C07328=1170.878,119.531,-53.606,-178.796,6.384,148.806
C07329=1170.873,119.780,-53.625,-178.793,6.386,148.805
C07330=1170.868,120.030,-53.645,-178.791,6.387,148.805
C07331=1170.864,120.279,-53.664,-178.789,6.388,148.804
C07332=1170.859,120.528,-53.683,-178.785,6.390,148.804
C07333=1170.854,120.778,-53.703,-178.783,6.391,148.803
C07334=1170.849,121.026,-53.722,-178.780,6.393,148.803
C07335=1170.844,121.276,-53.742,-178.777,6.395,148.803
C07336=1170.840,121.525,-53.761,-178.775,6.396,148.802
C07337=1170.835,121.774,-53.781,-178.772,6.397,148.802
C07338=1170.830,122.023,-53.800,-178.769,6.399,148.801
C07339=1170.826,122.273,-53.820,-178.766,6.401,148.801
C07340=1170.820,122.522,-53.839,-178.764,6.401,148.800
C07341=1170.816,122.771,-53.859,-178.761,6.403,148.800
C07342=1170.811,123.020,-53.878,-178.758,6.405,148.799
C07343=1170.806,123.269,-53.897,-178.756,6.406,148.799
C07344=1170.801,123.519,-53.917,-178.753,6.408,148.799
C07345=1170.796,123.767,-53.937,-178.751,6.409,148.798
C07346=1170.792,124.017,-53.957,-178.748,6.410,148.798
C07347=1170.787,124.266,-53.976,-178.745,6.412,148.797
C07348=1170.782,124.515,-53.995,-178.742,6.414,148.797
C07349=1170.778,124.764,-54.015,-178.740,6.415,148.796
C07350=1170.773,125.013,-54.035,-178.737,6.416,148.796
C07351=1170.768,125.263,-54.055,-178.734,6.418,148.795
C07352=1170.763,125.512,-54.074,-178.732,6.419,148.795
C07353=1170.758,125.761,-54.094,-178.729,6.421,148.795
C07354=1170.754,126.010,-54.114,-178.726,6.423,148.794
C07355=1170.749,126.259,-54.133,-178.723,6.425,148.794
C07356=1170.744,126.509,-54.153,-178.721,6.425,148.793
C07357=1170.739,126.758,-54.173,-178.718,6.427,148.793
C07358=1170.735,127.007,-54.193,-178.715,6.429,148.792
C07359=1170.729,127.256,-54.212,-178.713,6.430,148.792
C07360=1170.725,127.505,-54.233,-178.710,6.432,148.792
C07361=1170.720,127.755,-54.252,-178.708,6.433,148.791
C07362=1170.715,128.004,-54.272,-178.705,6.434,148.791
C07363=1170.710,128.252,-54.292,-178.702,6.436,148.790
C07364=1170.706,128.502,-54.312,-178.699,6.438,148.790
C07365=1170.701,128.752,-54.331,-178.697,6.440,148.789
C07366=1170.696,129.000,-54.352,-178.694,6.441,148.789
C07367=1170.691,129.249,-54.371,-178.692,6.442,148.789
C07368=1170.687,129.498,-54.391,-178.689,6.444,148.788
C07369=1170.682,129.748,-54.411,-178.686,6.445,148.788
C07370=1170.677,129.997,-54.431,-178.683,6.447,148.787
C07371=1170.672,130.246,-54.451,-178.680,6.449,148.787
C07372=1170.667,130.495,-54.470,-178.678,6.451,148.786
C07373=1170.663,130.744,-54.491,-178.675,6.452,148.786
C07374=1170.658,130.994,-54.510,-178.672,6.453,148.785
C07375=1170.654,131.243,-54.531,-178.670,6.455,148.785
C07376=1170.648,131.492,-54.550,-178.667,6.456,148.785
C07377=1170.643,131.741,-54.571,-178.664,6.458,148.784
C07378=1170.638,132.009,-54.592,-178.662,6.460,148.784
C07379=1170.633,132.278,-54.613,-178.658,6.461,148.783
C07380=1170.628,132.546,-54.635,-178.656,6.463,148.783
C07381=1170.623,132.815,-54.656,-178.653,6.465,148.782
C07382=1170.618,133.064,-54.677,-178.650,6.466,148.782
C07383=1170.613,133.314,-54.697,-178.647,6.468,148.781
C07384=1170.609,133.563,-54.717,-178.644,6.470,148.781
C07385=1170.604,133.812,-54.737,-178.642,6.471,148.781
C07386=1170.599,134.061,-54.757,-178.639,6.473,148.780
C07387=1170.595,134.310,-54.778,-178.637,6.474,148.780
C07388=1170.589,134.560,-54.798,-178.634,6.476,148.779
C07389=1170.585,134.809,-54.818,-178.631,6.477,148.779
C07390=1170.580,135.057,-54.839,-178.628,6.479,148.778
C07391=1170.575,135.307,-54.858,-178.626,6.481,148.778
C07392=1170.571,135.556,-54.879,-178.623,6.482,148.778
C07393=1170.566,135.805,-54.900,-178.620,6.484,148.777
C07394=1170.560,136.054,-54.919,-178.618,6.486,148.777
C07395=1170.556,136.303,-54.939,-178.615,6.488,148.776
C07396=1170.552,136.552,-54.960,-178.613,6.488,148.776
C07397=1170.546,136.802,-54.980,-178.610,6.490,148.775
C07398=1170.542,137.051,-55.000,-178.607,6.492,148.775
C07399=1170.537,137.300,-55.021,-178.604,6.493,148.775
C07400=1170.533,137.549,-55.041,-178.601,6.495,148.774
C07401=1170.528,137.798,-55.062,-178.599,6.497,148.774
C07402=1170.523,138.048,-55.082,-178.596,6.499,148.773
C07403=1170.518,138.296,-55.102,-178.593,6.500,148.773
C07404=1170.514,138.545,-55.122,-178.591,6.502,148.773
C07405=1170.509,138.795,-55.143,-178.588,6.503,148.772
C07406=1170.504,139.044,-55.164,-178.585,6.504,148.772
C07407=1170.500,139.293,-55.183,-178.583,6.506,148.771
C07408=1170.494,139.542,-55.204,-178.580,6.508,148.771
C07409=1170.489,139.791,-55.224,-178.577,6.510,148.771
C07410=1170.485,140.040,-55.245,-178.575,6.511,148.770
C07411=1170.480,140.289,-55.266,-178.572,6.513,148.770
C07412=1170.475,140.538,-55.286,-178.569,6.515,148.769
C07413=1170.471,140.787,-55.306,-178.566,6.517,148.769
C07414=1170.466,141.036,-55.327,-178.564,6.518,148.769
C07415=1170.461,141.286,-55.347,-178.561,6.520,148.768
C07416=1170.456,141.535,-55.368,-178.558,6.521,148.768
C07417=1170.451,141.784,-55.388,-178.556,6.522,148.767
C07418=1170.447,142.033,-55.409,-178.553,6.524,148.767
C07419=1170.442,142.282,-55.430,-178.550,6.526,148.766
C07420=1170.437,142.531,-55.450,-178.548,6.528,148.766
C07421=1170.432,142.780,-55.471,-178.545,6.529,148.766
C07422=1170.428,143.029,-55.491,-178.542,6.531,148.765
C07423=1170.424,143.279,-55.512,-178.540,6.533,148.765
C07424=1170.419,143.528,-55.533,-178.537,6.535,148.765
C07425=1170.414,143.777,-55.553,-178.534,6.536,148.764
C07426=1170.409,144.026,-55.574,-178.531,6.538,148.764
C07427=1170.405,144.275,-55.595,-178.528,6.539,148.763
C07428=1170.400,144.525,-55.616,-178.526,6.541,148.763
C07429=1170.395,144.773,-55.637,-178.523,6.543,148.762
C07430=1170.390,145.022,-55.658,-178.520,6.545,148.762
C07431=1170.386,145.271,-55.678,-178.517,6.546,148.762
C07432=1170.381,145.520,-55.699,-178.515,6.548,148.761
C07433=1170.376,145.769,-55.719,-178.513,6.549,148.761
C07434=1170.371,146.019,-55.740,-178.510,6.551,148.760
C07435=1170.367,146.268,-55.761,-178.507,6.553,148.760
C07436=1170.361,146.517,-55.782,-178.505,6.554,148.760
C07437=1170.357,146.765,-55.803,-178.502,6.556,148.759
C07438=1170.353,147.015,-55.824,-178.499,6.558,148.759
C07439=1170.348,147.264,-55.845,-178.496,6.560,148.759
C07440=1170.343,147.513,-55.866,-178.494,6.561,148.758
C07441=1170.338,147.763,-55.887,-178.491,6.563,148.758
C07442=1170.334,148.011,-55.908,-178.488,6.565,148.757
C07443=1170.329,148.260,-55.929,-178.485,6.566,148.757
C07444=1170.324,148.509,-55.949,-178.483,6.568,148.756
C07445=1170.319,148.758,-55.970,-178.480,6.570,148.756
C07446=1170.315,149.008,-55.992,-178.477,6.571,148.756
C07447=1170.310,149.257,-56.012,-178.474,6.573,148.755
C07448=1170.305,149.506,-56.033,-178.472,6.575,148.755
C07449=1170.301,149.755,-56.054,-178.469,6.577,148.754
C07450=1170.296,150.003,-56.075,-178.466,6.578,148.754
C07451=1170.291,150.253,-56.096,-178.464,6.580,148.754
C07452=1170.286,150.502,-56.117,-178.461,6.582,148.753
C07453=1170.282,150.751,-56.139,-178.458,6.584,148.753
C07454=1170.277,151.000,-56.160,-178.456,6.585,148.753
C07455=1170.272,151.249,-56.180,-178.453,6.587,148.752
C07456=1170.267,151.498,-56.202,-178.450,6.589,148.752
C07457=1170.262,151.747,-56.223,-178.447,6.591,148.751
C07458=1170.258,151.996,-56.245,-178.445,6.592,148.751
C07459=1170.254,152.245,-56.265,-178.442,6.594,148.751
C07460=1170.248,152.495,-56.286,-178.439,6.596,148.750
C07461=1170.244,152.743,-56.308,-178.437,6.598,148.750
C07462=1170.239,152.992,-56.328,-178.434,6.599,148.750
C07463=1170.235,153.242,-56.350,-178.431,6.601,148.749
C07464=1170.230,153.491,-56.371,-178.429,6.603,148.749
C07465=1170.225,153.740,-56.393,-178.426,6.605,148.748
C07466=1170.220,153.988,-56.413,-178.423,6.606,148.748
C07467=1170.216,154.238,-56.435,-178.421,6.608,148.748
C07468=1170.211,154.487,-56.456,-178.418,6.610,148.747
C07469=1170.206,154.736,-56.478,-178.415,6.612,148.747
C07470=1170.201,154.985,-56.499,-178.412,6.613,148.747
C07471=1170.197,155.234,-56.520,-178.410,6.615,148.746
C07472=1170.192,155.483,-56.541,-178.407,6.617,148.746
C07473=1170.187,155.732,-56.563,-178.404,6.619,148.745
C07474=1170.182,155.981,-56.584,-178.402,6.620,148.745
C07475=1170.178,156.230,-56.606,-178.399,6.622,148.745
C07476=1170.173,156.480,-56.627,-178.396,6.624,148.744
C07477=1170.169,156.728,-56.648,-178.394,6.626,148.744
C07478=1170.164,156.977,-56.670,-178.391,6.627,148.744
C07479=1170.159,157.227,-56.691,-178.388,6.629,148.743
C07480=1170.154,157.475,-56.713,-178.386,6.631,148.743
C07481=1170.149,157.724,-56.734,-178.383,6.633,148.742
C07482=1170.145,157.993,-56.757,-178.380,6.635,148.742
C07483=1170.139,158.262,-56.781,-178.377,6.637,148.742
C07484=1170.134,158.531,-56.803,-178.374,6.638,148.741
C07485=1170.129,158.800,-56.827,-178.371,6.640,148.741
C07486=1170.124,159.049,-56.848,-178.368,6.643,148.740
C07487=1170.120,159.299,-56.870,-178.365,6.644,148.740
C07488=1170.115,159.547,-56.892,-178.362,6.646,148.740
C07489=1170.111,159.796,-56.913,-178.360,6.648,148.739
C07490=1170.106,160.046,-56.935,-178.357,6.650,148.739
C07491=1170.101,160.294,-56.956,-178.355,6.652,148.739
C07492=1170.096,160.543,-56.978,-178.352,6.654,148.738
C07493=1170.092,160.792,-57.000,-178.349,6.655,148.738
C07494=1170.087,161.041,-57.022,-178.347,6.657,148.738
C07495=1170.083,161.291,-57.043,-178.344,6.659,148.737
C07496=1170.078,161.540,-57.065,-178.341,6.661,148.737
C07497=1170.073,161.788,-57.086,-178.339,6.662,148.736
C07498=1170.069,162.038,-57.108,-178.336,6.664,148.736
C07499=1170.064,162.286,-57.130,-178.333,6.666,148.736
C07500=1170.060,162.536,-57.152,-178.331,6.668,148.735
C07501=1170.054,162.785,-57.173,-178.328,6.669,148.735
C07502=1170.050,163.033,-57.195,-178.325,6.672,148.735
C07503=1170.045,163.283,-57.217,-178.322,6.674,148.734
C07504=1170.040,163.531,-57.238,-178.319,6.675,148.734
C07505=1170.036,163.781,-57.261,-178.317,6.677,148.733
C07506=1170.031,164.029,-57.282,-178.314,6.679,148.733
C07507=1170.026,164.279,-57.305,-178.311,6.681,148.733
C07508=1170.021,164.528,-57.327,-178.308,6.682,148.732
C07509=1170.016,164.776,-57.348,-178.306,6.684,148.732
C07510=1170.012,165.026,-57.370,-178.304,6.686,148.732
C07511=1170.007,165.274,-57.392,-178.301,6.688,148.731
C07512=1170.003,165.524,-57.414,-178.298,6.690,148.731
C07513=1169.998,165.772,-57.436,-178.296,6.692,148.731
C07514=1169.994,166.022,-57.458,-178.292,6.694,148.730
C07515=1169.989,166.270,-57.479,-178.290,6.696,148.730
C07516=1169.985,166.520,-57.501,-178.287,6.698,148.730
C07517=1169.979,166.769,-57.524,-178.284,6.699,148.729
C07518=1169.975,167.018,-57.546,-178.281,6.701,148.729
C07519=1169.970,167.267,-57.567,-178.279,6.703,148.729
C07520=1169.966,167.516,-57.590,-178.276,6.705,148.728
C07521=1169.961,167.765,-57.611,-178.273,6.706,148.728
C07522=1169.956,168.014,-57.634,-178.271,6.709,148.728
C07523=1169.951,168.262,-57.656,-178.268,6.711,148.727
C07524=1169.947,168.512,-57.678,-178.265,6.713,148.727
C07525=1169.942,168.760,-57.700,-178.263,6.715,148.727
C07526=1169.938,169.010,-57.722,-178.260,6.716,148.726
C07527=1169.932,169.258,-57.744,-178.257,6.718,148.726
C07528=1169.928,169.508,-57.766,-178.255,6.720,148.725
C07529=1169.924,169.756,-57.789,-178.252,6.722,148.725
C07530=1169.919,170.005,-57.811,-178.249,6.723,148.725
C07531=1169.914,170.254,-57.833,-178.246,6.726,148.724
C07532=1169.909,170.503,-57.855,-178.244,6.728,148.724
C07533=1169.905,170.752,-57.877,-178.241,6.730,148.724
C07534=1169.901,171.001,-57.900,-178.238,6.732,148.724
C07535=1169.896,171.250,-57.922,-178.236,6.733,148.723
C07536=1169.891,171.499,-57.944,-178.233,6.735,148.723
C07537=1169.887,171.748,-57.967,-178.230,6.737,148.722
C07538=1169.881,171.997,-57.989,-178.228,6.739,148.722
C07539=1169.877,172.246,-58.011,-178.224,6.741,148.722
C07540=1169.872,172.495,-58.033,-178.222,6.743,148.721
C07541=1169.867,172.744,-58.056,-178.219,6.745,148.721
C07542=1169.863,172.993,-58.078,-178.217,6.747,148.721
C07543=1169.858,173.242,-58.100,-178.214,6.749,148.720
C07544=1169.853,173.491,-58.123,-178.211,6.750,148.720
C07545=1169.849,173.740,-58.145,-178.209,6.752,148.720
C07546=1169.845,173.988,-58.168,-178.205,6.755,148.719
C07547=1169.840,174.238,-58.190,-178.203,6.757,148.719
C07548=1169.835,174.486,-58.212,-178.201,6.759,148.719
C07549=1169.830,174.735,-58.235,-178.198,6.760,148.719
C07550=1169.826,174.985,-58.257,-178.195,6.762,148.718
C07551=1169.821,175.233,-58.280,-178.192,6.764,148.718
C07552=1169.816,175.483,-58.302,-178.189,6.767,148.717
C07553=1169.812,175.731,-58.325,-178.187,6.768,148.717
C07554=1169.807,175.980,-58.347,-178.184,6.770,148.717
C07555=1169.803,176.229,-58.370,-178.182,6.772,148.717
C07556=1169.798,176.479,-58.393,-178.179,6.774,148.716
C07557=1169.793,176.727,-58.415,-178.176,6.776,148.716
C07558=1169.789,176.976,-58.437,-178.173,6.778,148.715
C07559=1169.784,177.225,-58.461,-178.170,6.780,148.715
C07560=1169.779,177.474,-58.482,-178.168,6.782,148.715
C07561=1169.775,177.723,-58.506,-178.165,6.784,148.715
C07562=1169.770,177.972,-58.528,-178.163,6.786,148.714
C07563=1169.765,178.220,-58.551,-178.160,6.788,148.714
C07564=1169.761,178.469,-58.573,-178.157,6.790,148.714
C07565=1169.756,178.719,-58.596,-178.154,6.792,148.713
C07566=1169.752,178.967,-58.619,-178.151,6.794,148.713
C07567=1169.746,179.216,-58.641,-178.149,6.796,148.713
C07568=1169.742,179.465,-58.664,-178.147,6.797,148.712
C07569=1169.738,179.714,-58.687,-178.143,6.800,148.712
C07570=1169.733,179.964,-58.710,-178.141,6.802,148.712
C07571=1169.728,180.212,-58.732,-178.138,6.804,148.711
C07572=1169.724,180.461,-58.756,-178.135,6.805,148.711
C07573=1169.719,180.710,-58.778,-178.133,6.807,148.711
C07574=1169.715,180.959,-58.801,-178.130,6.810,148.710
C07575=1169.710,181.207,-58.823,-178.127,6.812,148.710
C07576=1169.705,181.456,-58.847,-178.124,6.814,148.710
C07577=1169.700,181.706,-58.869,-178.122,6.815,148.709
C07578=1169.696,181.955,-58.892,-178.119,6.818,148.709
C07579=1169.691,182.203,-58.915,-178.116,6.820,148.709
C07580=1169.687,182.452,-58.938,-178.114,6.822,148.709
C07581=1169.682,182.701,-58.961,-178.111,6.824,148.708
C07582=1169.677,182.950,-58.984,-178.108,6.825,148.708
C07583=1169.673,183.199,-59.007,-178.105,6.828,148.708
C07584=1169.669,183.448,-59.030,-178.103,6.830,148.707
C07585=1169.663,183.696,-59.053,-178.100,6.832,148.707
C07586=1169.659,183.966,-59.078,-178.097,6.834,148.707
C07587=1169.653,184.236,-59.103,-178.094,6.836,148.706
C07588=1169.648,184.505,-59.128,-178.091,6.839,148.706
C07589=1169.644,184.775,-59.152,-178.088,6.840,148.706
C07590=1169.639,185.024,-59.175,-178.086,6.843,148.705
C07591=1169.634,185.273,-59.199,-178.083,6.845,148.705
C07592=1169.629,185.522,-59.222,-178.080,6.847,148.705
C07593=1169.626,185.771,-59.245,-178.077,6.849,148.704
C07594=1169.621,186.020,-59.268,-178.075,6.850,148.704
C07595=1169.616,186.269,-59.292,-178.073,6.853,148.704
C07596=1169.611,186.517,-59.315,-178.069,6.855,148.704
C07597=1169.607,186.766,-59.337,-178.067,6.857,148.703
C07598=1169.602,187.015,-59.361,-178.064,6.859,148.703
C07599=1169.597,187.264,-59.384,-178.062,6.861,148.703
C07600=1169.593,187.513,-59.407,-178.058,6.863,148.702
C07601=1169.589,187.762,-59.430,-178.056,6.865,148.702
C07602=1169.584,188.011,-59.454,-178.053,6.867,148.702
C07603=1169.579,188.260,-59.477,-178.051,6.869,148.702
C07604=1169.575,188.509,-59.500,-178.048,6.872,148.701
C07605=1169.569,188.757,-59.523,-178.045,6.873,148.701
C07606=1169.565,189.006,-59.547,-178.042,6.875,148.701
C07607=1169.561,189.255,-59.569,-178.040,6.878,148.700
C07608=1169.556,189.504,-59.593,-178.037,6.880,148.700
C07609=1169.552,189.752,-59.617,-178.034,6.882,148.700
C07610=1169.547,190.001,-59.640,-178.032,6.883,148.699
C07611=1169.542,190.250,-59.664,-178.029,6.886,148.699
C07612=1169.538,190.499,-59.687,-178.026,6.888,148.699
C07613=1169.533,190.748,-59.710,-178.023,6.890,148.699
C07614=1169.528,190.997,-59.734,-178.021,6.892,148.698
C07615=1169.523,191.246,-59.757,-178.018,6.895,148.698
C07616=1169.520,191.495,-59.780,-178.015,6.896,148.698
C07617=1169.515,191.744,-59.804,-178.013,6.898,148.697
C07618=1169.510,191.993,-59.827,-178.010,6.901,148.697
C07619=1169.506,192.242,-59.851,-178.007,6.903,148.697
C07620=1169.501,192.490,-59.875,-178.004,6.905,148.697
C07621=1169.497,192.739,-59.898,-178.002,6.906,148.696
C07622=1169.492,192.988,-59.921,-177.999,6.909,148.696
C07623=1169.487,193.237,-59.945,-177.996,6.911,148.696
C07624=1169.483,193.486,-59.969,-177.994,6.913,148.695
C07625=1169.478,193.735,-59.992,-177.991,6.916,148.695
C07626=1169.473,193.984,-60.015,-177.988,6.918,148.695
C07627=1169.469,194.232,-60.040,-177.986,6.919,148.695
C07628=1169.464,194.481,-60.063,-177.983,6.921,148.694
C07629=1169.460,194.730,-60.086,-177.980,6.924,148.694
C07630=1169.455,194.978,-60.110,-177.977,6.926,148.694
C07631=1169.451,195.228,-60.134,-177.975,6.928,148.693
C07632=1169.446,195.476,-60.158,-177.972,6.931,148.693
C07633=1169.441,195.725,-60.181,-177.969,6.932,148.693
C07634=1169.437,195.974,-60.204,-177.967,6.934,148.693
C07635=1169.432,196.222,-60.229,-177.964,6.937,148.692
C07636=1169.427,196.472,-60.253,-177.961,6.939,148.692
C07637=1169.422,196.720,-60.277,-177.958,6.941,148.692
C07638=1169.418,196.969,-60.300,-177.955,6.943,148.691
C07639=1169.413,197.218,-60.324,-177.953,6.945,148.691
C07640=1169.409,197.467,-60.347,-177.950,6.947,148.691
C07641=1169.405,197.716,-60.372,-177.947,6.950,148.691
C07642=1169.400,197.965,-60.395,-177.945,6.952,148.691
C07643=1169.396,198.213,-60.419,-177.942,6.954,148.690
C07644=1169.391,198.462,-60.443,-177.939,6.956,148.690
C07645=1169.386,198.711,-60.467,-177.937,6.958,148.690
C07646=1169.381,198.960,-60.491,-177.934,6.960,148.689
C07647=1169.377,199.208,-60.515,-177.931,6.963,148.689
C07648=1169.372,199.457,-60.538,-177.929,6.965,148.689
C07649=1169.368,199.706,-60.562,-177.926,6.967,148.689
C07650=1169.364,199.955,-60.587,-177.923,6.969,148.688
C07651=1169.359,200.204,-60.611,-177.921,6.971,148.688
C07652=1169.354,200.453,-60.635,-177.918,6.973,148.688
C07653=1169.350,200.701,-60.659,-177.915,6.976,148.687
C07654=1169.345,200.950,-60.682,-177.912,6.978,148.687
C07655=1169.341,201.199,-60.706,-177.910,6.980,148.687
C07656=1169.336,201.448,-60.731,-177.907,6.982,148.687
C07657=1169.331,201.697,-60.755,-177.904,6.984,148.687
C07658=1169.327,201.945,-60.779,-177.902,6.986,148.686
C07659=1169.323,202.194,-60.803,-177.899,6.989,148.686
C07660=1169.317,202.443,-60.827,-177.896,6.991,148.686
C07661=1169.313,202.692,-60.851,-177.894,6.993,148.685
C07662=1169.309,202.941,-60.875,-177.891,6.996,148.685
C07663=1169.305,203.189,-60.899,-177.888,6.997,148.685
C07664=1169.299,203.438,-60.923,-177.885,7.000,148.685
C07665=1169.295,203.687,-60.947,-177.883,7.002,148.685
C07666=1169.290,203.935,-60.971,-177.880,7.004,148.684
C07667=1169.286,204.185,-60.996,-177.877,7.007,148.684
C07668=1169.281,204.433,-61.020,-177.875,7.009,148.684
C07669=1169.277,204.682,-61.045,-177.872,7.010,148.683
C07670=1169.272,204.931,-61.068,-177.869,7.013,148.683
C07671=1169.268,205.180,-61.093,-177.866,7.015,148.683
C07672=1169.263,205.428,-61.117,-177.863,7.018,148.683
C07673=1169.258,205.677,-61.142,-177.861,7.020,148.682
C07674=1169.254,205.926,-61.166,-177.858,7.022,148.682
C07675=1169.249,206.175,-61.191,-177.856,7.024,148.682
C07676=1169.245,206.423,-61.215,-177.853,7.026,148.682
C07677=1169.241,206.672,-61.239,-177.850,7.028,148.681
C07678=1169.236,206.921,-61.264,-177.847,7.031,148.681
C07679=1169.232,207.170,-61.288,-177.845,7.033,148.681
C07680=1169.226,207.419,-61.312,-177.842,7.036,148.681
C07681=1169.222,207.667,-61.336,-177.839,7.037,148.680
C07682=1169.217,207.917,-61.361,-177.837,7.039,148.680
C07683=1169.213,208.165,-61.385,-177.834,7.042,148.680
C07684=1169.209,208.414,-61.409,-177.831,7.044,148.680
C07685=1169.204,208.662,-61.435,-177.828,7.047,148.680
C07686=1169.200,208.911,-61.459,-177.826,7.049,148.679
C07687=1169.195,209.160,-61.484,-177.823,7.050,148.679
C07688=1169.190,209.408,-61.508,-177.820,7.053,148.679
C07689=1169.186,209.657,-61.533,-177.818,7.055,148.678
C07690=1169.181,209.928,-61.560,-177.815,7.058,148.678
C07691=1169.175,210.198,-61.586,-177.812,7.061,148.678
C07692=1169.171,210.469,-61.613,-177.809,7.063,148.678
C07693=1169.166,210.739,-61.639,-177.806,7.065,148.677
C07694=1169.162,210.989,-61.664,-177.803,7.068,148.677
C07695=1169.157,211.237,-61.689,-177.800,7.070,148.677
C07696=1169.153,211.485,-61.713,-177.798,7.072,148.677
C07697=1169.148,211.735,-61.738,-177.795,7.075,148.677
C07698=1169.143,211.983,-61.763,-177.793,7.077,148.676
C07699=1169.138,212.232,-61.787,-177.789,7.079,148.676
C07700=1169.134,212.480,-61.813,-177.787,7.081,148.676
C07701=1169.130,212.729,-61.837,-177.784,7.084,148.676
C07702=1169.125,212.978,-61.862,-177.781,7.086,148.675
C07703=1169.121,213.227,-61.886,-177.779,7.088,148.675
C07704=1169.116,213.475,-61.911,-177.776,7.091,148.675
C07705=1169.112,213.724,-61.936,-177.774,7.093,148.675
C07706=1169.107,213.973,-61.960,-177.770,7.095,148.674
C07707=1169.103,214.222,-61.985,-177.768,7.097,148.674
C07708=1169.098,214.470,-62.011,-177.765,7.100,148.674
C07709=1169.093,214.719,-62.035,-177.763,7.102,148.674
C07710=1169.089,214.968,-62.060,-177.760,7.105,148.674
C07711=1169.084,215.216,-62.085,-177.757,7.107,148.674
C07712=1169.080,215.465,-62.110,-177.755,7.109,148.673
C07713=1169.075,215.714,-62.134,-177.752,7.111,148.673
C07714=1169.071,215.963,-62.160,-177.749,7.113,148.673
C07715=1169.067,216.211,-62.184,-177.746,7.116,148.672
C07716=1169.062,216.460,-62.210,-177.744,7.118,148.672
C07717=1169.057,216.709,-62.235,-177.741,7.121,148.672
C07718=1169.053,216.958,-62.260,-177.738,7.123,148.672
C07719=1169.049,217.206,-62.285,-177.735,7.125,148.672
C07720=1169.044,217.455,-62.310,-177.733,7.128,148.671
C07721=1169.039,217.703,-62.335,-177.730,7.130,148.671
C07722=1169.035,217.953,-62.360,-177.728,7.132,148.671
C07723=1169.031,218.201,-62.385,-177.724,7.135,148.671
C07724=1169.026,218.450,-62.410,-177.722,7.137,148.671
C07725=1169.021,218.698,-62.435,-177.719,7.140,148.670
C07726=1169.017,218.948,-62.460,-177.717,7.142,148.670
C07727=1169.012,219.196,-62.486,-177.714,7.144,148.670
C07728=1169.008,219.445,-62.510,-177.711,7.147,148.670
C07729=1169.003,219.693,-62.535,-177.709,7.148,148.669
C07730=1168.999,219.942,-62.561,-177.706,7.151,148.669
C07731=1168.994,220.190,-62.586,-177.703,7.153,148.669
C07732=1168.990,220.439,-62.612,-177.700,7.156,148.669
C07733=1168.985,220.688,-62.636,-177.698,7.158,148.669
C07734=1168.981,220.936,-62.661,-177.695,7.161,148.669
C07735=1168.977,221.185,-62.687,-177.692,7.163,148.668
C07736=1168.972,221.434,-62.712,-177.690,7.165,148.668
C07737=1168.967,221.683,-62.738,-177.687,7.167,148.668
C07738=1168.963,221.931,-62.763,-177.684,7.170,148.668
C07739=1168.958,222.180,-62.788,-177.681,7.172,148.667
C07740=1168.953,222.428,-62.813,-177.679,7.175,148.667
C07741=1168.949,222.677,-62.839,-177.677,7.177,148.667
C07742=1168.945,222.926,-62.865,-177.673,7.180,148.667
C07743=1168.940,223.175,-62.890,-177.671,7.182,148.667
C07744=1168.936,223.423,-62.915,-177.668,7.184,148.666
C07745=1168.931,223.671,-62.940,-177.666,7.187,148.666
C07746=1168.927,223.920,-62.966,-177.662,7.189,148.666
C07747=1168.923,224.170,-62.991,-177.660,7.192,148.666
C07748=1168.918,224.418,-63.016,-177.657,7.194,148.666
C07749=1168.914,224.666,-63.042,-177.654,7.197,148.665
C07750=1168.909,224.915,-63.068,-177.652,7.199,148.665
C07751=1168.905,225.163,-63.093,-177.649,7.202,148.665
C07752=1168.900,225.412,-63.119,-177.647,7.204,148.665
C07753=1168.896,225.662,-63.144,-177.643,7.206,148.665
C07754=1168.891,225.910,-63.169,-177.641,7.208,148.665
C07755=1168.887,226.159,-63.195,-177.638,7.211,148.664
C07756=1168.883,226.407,-63.221,-177.636,7.213,148.664
C07757=1168.877,226.656,-63.247,-177.633,7.216,148.664
C07758=1168.873,226.905,-63.273,-177.630,7.218,148.664
C07759=1168.869,227.153,-63.298,-177.628,7.221,148.664
C07760=1168.864,227.401,-63.324,-177.625,7.223,148.663
C07761=1168.859,227.650,-63.349,-177.622,7.226,148.663
C07762=1168.855,227.899,-63.375,-177.619,7.228,148.663
C07763=1168.850,228.147,-63.401,-177.617,7.230,148.663
C07764=1168.846,228.396,-63.426,-177.614,7.233,148.663
C07765=1168.842,228.645,-63.452,-177.611,7.235,148.662
C07766=1168.838,228.894,-63.478,-177.609,7.238,148.662
C07767=1168.832,229.142,-63.504,-177.606,7.240,148.662
C07768=1168.828,229.391,-63.530,-177.603,7.243,148.662
C07769=1168.824,229.640,-63.555,-177.600,7.245,148.662
C07770=1168.819,229.888,-63.581,-177.598,7.248,148.662
C07771=1168.815,230.137,-63.606,-177.595,7.251,148.661
C07772=1168.810,230.385,-63.632,-177.592,7.252,148.661
C07773=1168.806,230.634,-63.658,-177.590,7.255,148.661
C07774=1168.801,230.883,-63.684,-177.587,7.257,148.661
C07775=1168.797,231.131,-63.710,-177.584,7.260,148.661
C07776=1168.793,231.380,-63.736,-177.582,7.262,148.661
C07777=1168.788,231.628,-63.762,-177.579,7.265,148.660
C07778=1168.783,231.877,-63.788,-177.576,7.268,148.660
C07779=1168.778,232.126,-63.814,-177.574,7.270,148.660
C07780=1168.774,232.374,-63.839,-177.571,7.272,148.660
C07781=1168.770,232.623,-63.866,-177.568,7.275,148.660
C07782=1168.765,232.872,-63.892,-177.565,7.277,148.659
C07783=1168.761,233.120,-63.918,-177.563,7.279,148.659
C07784=1168.756,233.369,-63.943,-177.560,7.282,148.659
C07785=1168.752,233.617,-63.970,-177.557,7.285,148.659
C07786=1168.747,233.866,-63.996,-177.555,7.287,148.659
C07787=1168.743,234.115,-64.022,-177.552,7.290,148.659
C07788=1168.739,234.364,-64.048,-177.549,7.292,148.658
C07789=1168.734,234.612,-64.075,-177.547,7.295,148.658
C07790=1168.730,234.860,-64.100,-177.544,7.298,148.658
C07791=1168.725,235.109,-64.126,-177.541,7.299,148.658
C07792=1168.721,235.357,-64.153,-177.538,7.302,148.658
C07793=1168.716,235.606,-64.179,-177.536,7.305,148.658
C07794=1168.712,235.877,-64.207,-177.533,7.307,148.657
C07795=1168.707,236.150,-64.236,-177.530,7.310,148.657
C07796=1168.702,236.421,-64.265,-177.527,7.313,148.657
C07797=1168.698,236.693,-64.293,-177.524,7.316,148.657
C07798=1168.693,236.941,-64.320,-177.521,7.318,148.657
C07799=1168.688,237.189,-64.345,-177.519,7.320,148.657
C07800=1168.683,237.438,-64.372,-177.516,7.323,148.656
C07801=1168.679,237.687,-64.398,-177.513,7.326,148.656
C07802=1168.675,237.935,-64.425,-177.511,7.328,148.656
C07803=1168.670,238.184,-64.451,-177.508,7.331,148.656
C07804=1168.666,238.432,-64.477,-177.505,7.334,148.656
C07805=1168.661,238.681,-64.504,-177.502,7.336,148.656
C07806=1168.657,238.930,-64.530,-177.500,7.339,148.656
C07807=1168.653,239.179,-64.557,-177.498,7.341,148.655
C07808=1168.649,239.427,-64.583,-177.494,7.344,148.655
C07809=1168.644,239.676,-64.609,-177.492,7.347,148.655
C07810=1168.640,239.924,-64.636,-177.489,7.349,148.655
C07811=1168.635,240.173,-64.662,-177.487,7.352,148.655
C07812=1168.630,240.421,-64.688,-177.483,7.354,148.655
C07813=1168.626,240.669,-64.715,-177.481,7.356,148.655
C07814=1168.621,240.918,-64.741,-177.478,7.359,148.654
C07815=1168.617,241.167,-64.768,-177.475,7.362,148.654
C07816=1168.613,241.415,-64.795,-177.473,7.364,148.654
C07817=1168.608,241.664,-64.821,-177.470,7.367,148.654
C07818=1168.603,241.912,-64.848,-177.467,7.370,148.654
C07819=1168.599,242.161,-64.875,-177.465,7.372,148.654
C07820=1168.594,242.410,-64.901,-177.462,7.375,148.654
C07821=1168.590,242.658,-64.927,-177.459,7.378,148.653
C07822=1168.586,242.906,-64.954,-177.457,7.380,148.653
C07823=1168.582,243.155,-64.981,-177.454,7.382,148.653
C07824=1168.577,243.404,-65.007,-177.452,7.385,148.653
C07825=1168.572,243.652,-65.034,-177.449,7.388,148.653
C07826=1168.568,243.900,-65.061,-177.446,7.390,148.653
C07827=1168.564,244.149,-65.088,-177.444,7.392,148.653
C07828=1168.559,244.397,-65.115,-177.441,7.395,148.652
C07829=1168.555,244.647,-65.141,-177.438,7.398,148.652
C07830=1168.551,244.895,-65.168,-177.435,7.401,148.652
C07831=1168.546,245.144,-65.195,-177.433,7.403,148.652
C07832=1168.542,245.392,-65.222,-177.430,7.406,148.652
C07833=1168.537,245.640,-65.249,-177.427,7.409,148.652
C07834=1168.533,245.889,-65.276,-177.425,7.411,148.652
C07835=1168.529,246.137,-65.302,-177.422,7.414,148.651
C07836=1168.524,246.386,-65.328,-177.419,7.417,148.651
C07837=1168.519,246.635,-65.356,-177.417,7.419,148.651
C07838=1168.515,246.883,-65.382,-177.414,7.422,148.651
C07839=1168.511,247.131,-65.409,-177.411,7.425,148.651
C07840=1168.506,247.380,-65.436,-177.409,7.426,148.651
C07841=1168.501,247.628,-65.463,-177.406,7.429,148.651
C07842=1168.498,247.877,-65.490,-177.403,7.432,148.651
C07843=1168.493,248.126,-65.517,-177.401,7.434,148.651
C07844=1168.489,248.374,-65.544,-177.398,7.437,148.651
C07845=1168.484,248.623,-65.571,-177.395,7.440,148.650
C07846=1168.479,248.871,-65.598,-177.392,7.443,148.650
C07847=1168.475,249.120,-65.625,-177.390,7.445,148.650
C07848=1168.471,249.368,-65.652,-177.387,7.448,148.650
C07849=1168.466,249.616,-65.679,-177.384,7.451,148.650
C07850=1168.462,249.865,-65.707,-177.382,7.453,148.650
C07851=1168.458,250.114,-65.734,-177.379,7.456,148.650
C07852=1168.454,250.362,-65.761,-177.376,7.459,148.650
C07853=1168.449,250.610,-65.788,-177.374,7.461,148.649
C07854=1168.445,250.859,-65.815,-177.371,7.464,148.649
C07855=1168.440,251.107,-65.842,-177.369,7.467,148.649
C07856=1168.436,251.356,-65.869,-177.365,7.469,148.649
C07857=1168.431,251.604,-65.897,-177.363,7.472,148.649
C07858=1168.427,251.853,-65.924,-177.360,7.475,148.649
C07859=1168.422,252.101,-65.951,-177.358,7.478,148.649
C07860=1168.418,252.349,-65.978,-177.355,7.480,148.649
C07861=1168.414,252.599,-66.005,-177.353,7.483,148.649
C07862=1168.410,252.847,-66.033,-177.350,7.485,148.648
C07863=1168.405,253.095,-66.060,-177.347,7.488,148.648
C07864=1168.401,253.344,-66.087,-177.345,7.490,148.648
C07865=1168.396,253.593,-66.114,-177.342,7.493,148.648
C07866=1168.392,253.841,-66.142,-177.339,7.496,148.648
C07867=1168.387,254.089,-66.169,-177.336,7.499,148.648
C07868=1168.383,254.338,-66.196,-177.334,7.501,148.648
C07869=1168.379,254.586,-66.224,-177.331,7.504,148.648
C07870=1168.374,254.835,-66.251,-177.328,7.507,148.648
C07871=1168.370,255.083,-66.278,-177.325,7.510,148.648
C07872=1168.365,255.331,-66.306,-177.323,7.512,148.647
C07873=1168.361,255.580,-66.334,-177.320,7.515,148.647
C07874=1168.357,255.828,-66.361,-177.318,7.518,148.647
C07875=1168.352,256.077,-66.388,-177.315,7.521,148.647
C07876=1168.348,256.325,-66.416,-177.313,7.523,148.647
C07877=1168.344,256.574,-66.444,-177.310,7.526,148.647
C07878=1168.339,256.822,-66.471,-177.307,7.529,148.647
C07879=1168.335,257.070,-66.499,-177.304,7.532,148.647
C07880=1168.331,257.319,-66.526,-177.302,7.534,148.647
C07881=1168.326,257.567,-66.554,-177.299,7.537,148.647
C07882=1168.321,257.816,-66.581,-177.296,7.540,148.647
C07883=1168.317,258.065,-66.610,-177.294,7.543,148.646
C07884=1168.313,258.313,-66.637,-177.291,7.545,148.646
C07885=1168.308,258.561,-66.664,-177.289,7.548,148.646
C07886=1168.304,258.810,-66.692,-177.286,7.551,148.646
C07887=1168.300,259.058,-66.720,-177.283,7.554,148.646
C07888=1168.296,259.306,-66.747,-177.281,7.555,148.646
C07889=1168.291,259.555,-66.775,-177.278,7.558,148.646
C07890=1168.286,259.803,-66.803,-177.275,7.561,148.646
C07891=1168.282,260.052,-66.830,-177.272,7.564,148.646
C07892=1168.278,260.300,-66.858,-177.269,7.567,148.646
C07893=1168.274,260.548,-66.886,-177.267,7.569,148.646
C07894=1168.269,260.797,-66.913,-177.265,7.572,148.646
C07895=1168.265,261.046,-66.942,-177.262,7.575,148.645
C07896=1168.260,261.293,-66.970,-177.259,7.578,148.645
C07897=1168.256,261.543,-66.997,-177.257,7.580,148.645
C07898=1168.251,261.815,-67.027,-177.254,7.584,148.645
C07899=1168.246,262.089,-67.058,-177.251,7.587,148.645
C07900=1168.242,262.361,-67.090,-177.248,7.590,148.645
C07901=1168.237,262.635,-67.120,-177.245,7.593,148.645
C07902=1168.233,262.883,-67.147,-177.242,7.596,148.645
C07903=1168.228,263.132,-67.176,-177.239,7.599,148.645
C07904=1168.224,263.380,-67.204,-177.237,7.602,148.645
C07905=1168.219,263.628,-67.232,-177.234,7.604,148.645
C07906=1168.216,263.876,-67.260,-177.232,7.607,148.645
C07907=1168.210,264.125,-67.287,-177.229,7.610,148.645
C07908=1168.206,264.374,-67.315,-177.226,7.613,148.645
C07909=1168.202,264.622,-67.343,-177.223,7.616,148.644
C07910=1168.198,264.870,-67.372,-177.221,7.618,148.644
C07911=1168.193,265.118,-67.400,-177.218,7.621,148.644
C07912=1168.189,265.367,-67.429,-177.216,7.624,148.644
C07913=1168.184,265.615,-67.456,-177.213,7.627,148.644
C07914=1168.181,265.864,-67.484,-177.210,7.630,148.644
C07915=1168.176,266.112,-67.513,-177.208,7.632,148.644
C07916=1168.171,266.360,-67.541,-177.205,7.635,148.644
C07917=1168.167,266.609,-67.568,-177.203,7.638,148.644
C07918=1168.162,266.857,-67.596,-177.200,7.641,148.644
C07919=1168.158,267.106,-67.625,-177.197,7.644,148.644
C07920=1168.154,267.355,-67.653,-177.195,7.646,148.644
C07921=1168.149,267.602,-67.681,-177.192,7.649,148.644
C07922=1168.145,267.851,-67.710,-177.189,7.652,148.644
C07923=1168.141,268.099,-67.738,-177.187,7.655,148.644
C07924=1168.137,268.347,-67.766,-177.184,7.658,148.644
C07925=1168.132,268.595,-67.795,-177.181,7.661,148.644
C07926=1168.128,268.844,-67.823,-177.179,7.663,148.643
C07927=1168.123,269.092,-67.851,-177.176,7.666,148.643
C07928=1168.120,269.341,-67.879,-177.173,7.669,148.643
C07929=1168.114,269.589,-67.908,-177.171,7.672,148.643
C07930=1168.111,269.837,-67.936,-177.168,7.675,148.643
C07931=1168.106,270.086,-67.964,-177.165,7.678,148.643
C07932=1168.102,270.334,-67.992,-177.163,7.680,148.643
C07933=1168.098,270.583,-68.022,-177.160,7.683,148.643
C07934=1168.093,270.830,-68.050,-177.157,7.686,148.643
C07935=1168.089,271.079,-68.078,-177.155,7.689,148.643
C07936=1168.084,271.327,-68.107,-177.152,7.692,148.643
C07937=1168.080,271.576,-68.135,-177.150,7.695,148.643
C07938=1168.076,271.824,-68.164,-177.147,7.698,148.643
C07939=1168.071,272.072,-68.192,-177.145,7.700,148.643
C07940=1168.067,272.321,-68.221,-177.142,7.703,148.643
C07941=1168.063,272.569,-68.249,-177.139,7.706,148.643
C07942=1168.058,272.817,-68.278,-177.136,7.709,148.643
C07943=1168.054,273.066,-68.307,-177.134,7.712,148.643
C07944=1168.050,273.314,-68.335,-177.131,7.715,148.643
C07945=1168.045,273.562,-68.364,-177.128,7.718,148.643
C07946=1168.041,273.811,-68.393,-177.126,7.720,148.643
C07947=1168.037,274.059,-68.421,-177.123,7.723,148.643
C07948=1168.032,274.307,-68.450,-177.121,7.726,148.642
C07949=1168.028,274.556,-68.479,-177.118,7.729,148.642
C07950=1168.024,274.803,-68.507,-177.116,7.732,148.643
C07951=1168.019,275.052,-68.536,-177.113,7.735,148.643
C07952=1168.015,275.301,-68.565,-177.110,7.738,148.643
C07953=1168.011,275.548,-68.593,-177.108,7.740,148.642
C07954=1168.006,275.797,-68.622,-177.105,7.743,148.642
C07955=1168.002,276.046,-68.651,-177.102,7.746,148.642
C07956=1167.998,276.294,-68.680,-177.100,7.749,148.642
C07957=1167.994,276.542,-68.709,-177.097,7.752,148.642
C07958=1167.989,276.791,-68.737,-177.094,7.755,148.642
C07959=1167.985,277.039,-68.767,-177.092,7.758,148.642
C07960=1167.981,277.287,-68.795,-177.089,7.761,148.642
C07961=1167.976,277.535,-68.824,-177.087,7.763,148.642
C07962=1167.972,277.784,-68.853,-177.084,7.766,148.642
C07963=1167.968,278.032,-68.882,-177.081,7.769,148.642
C07964=1167.963,278.280,-68.910,-177.079,7.772,148.642
C07965=1167.959,278.528,-68.940,-177.076,7.775,148.642
C07966=1167.955,278.777,-68.969,-177.073,7.778,148.642
C07967=1167.951,279.026,-68.998,-177.071,7.782,148.642
C07968=1167.946,279.273,-69.027,-177.068,7.784,148.642
C07969=1167.942,279.521,-69.056,-177.065,7.787,148.642
C07970=1167.938,279.770,-69.084,-177.063,7.790,148.642
C07971=1167.934,280.018,-69.114,-177.060,7.793,148.642
C07972=1167.930,280.266,-69.143,-177.058,7.796,148.642
C07973=1167.924,280.515,-69.172,-177.055,7.798,148.642
C07974=1167.920,280.763,-69.201,-177.053,7.802,148.642
C07975=1167.916,281.011,-69.231,-177.050,7.805,148.642
C07976=1167.912,281.260,-69.259,-177.047,7.808,148.642
C07977=1167.908,281.508,-69.288,-177.044,7.811,148.642
C07978=1167.903,281.756,-69.317,-177.042,7.814,148.642
C07979=1167.899,282.004,-69.347,-177.039,7.817,148.642
C07980=1167.895,282.252,-69.376,-177.037,7.820,148.642
C07981=1167.890,282.501,-69.405,-177.034,7.822,148.642
C07982=1167.886,282.749,-69.434,-177.032,7.825,148.642
C07983=1167.882,282.997,-69.463,-177.029,7.828,148.642
C07984=1167.877,283.245,-69.493,-177.026,7.831,148.642
C07985=1167.873,283.493,-69.522,-177.023,7.834,148.642
C07986=1167.869,283.742,-69.552,-177.021,7.837,148.642
C07987=1167.864,283.991,-69.581,-177.018,7.840,148.642
C07988=1167.860,284.239,-69.610,-177.016,7.843,148.642
C07989=1167.856,284.487,-69.639,-177.013,7.846,148.642
C07990=1167.851,284.735,-69.669,-177.010,7.849,148.642
C07991=1167.847,284.983,-69.698,-177.008,7.852,148.642
C07992=1167.843,285.231,-69.727,-177.005,7.855,148.642
C07993=1167.839,285.479,-69.757,-177.003,7.857,148.642
C07994=1167.835,285.728,-69.786,-177.000,7.860,148.642
C07995=1167.830,285.976,-69.816,-176.997,7.863,148.642
C07996=1167.826,286.224,-69.845,-176.995,7.867,148.642
C07997=1167.822,286.472,-69.875,-176.992,7.870,148.642
C07998=1167.818,286.721,-69.904,-176.990,7.873,148.642
C07999=1167.813,286.969,-69.934,-176.987,7.876,148.642
C08000=1167.809,287.218,-69.964,-176.984,7.879,148.642
C08001=1167.804,287.465,-69.993,-176.982,7.882,148.642
C08002=1167.799,287.740,-70.026,-176.979,7.885,148.642
C08003=1167.795,288.015,-70.058,-176.976,7.889,148.642
C08004=1167.791,288.290,-70.091,-176.973,7.892,148.642
C08005=1167.786,288.565,-70.124,-176.970,7.895,148.642
C08006=1167.781,288.813,-70.153,-176.968,7.898,148.642
C08007=1167.777,289.062,-70.183,-176.965,7.901,148.642
C08008=1167.773,289.309,-70.213,-176.963,7.904,148.642
C08009=1167.768,289.558,-70.243,-176.960,7.907,148.642
C08010=1167.764,289.806,-70.273,-176.958,7.910,148.642
C08011=1167.760,290.054,-70.302,-176.955,7.913,148.642
C08012=1167.756,290.303,-70.332,-176.952,7.916,148.642
C08013=1167.752,290.550,-70.362,-176.949,7.919,148.642
C08014=1167.747,290.799,-70.392,-176.947,7.922,148.642
C08015=1167.743,291.047,-70.421,-176.944,7.925,148.642
C08016=1167.739,291.295,-70.451,-176.942,7.928,148.642
C08017=1167.735,291.543,-70.481,-176.939,7.931,148.642
C08018=1167.730,291.792,-70.511,-176.937,7.934,148.642
C08019=1167.726,292.040,-70.540,-176.934,7.937,148.642
C08020=1167.722,292.288,-70.570,-176.931,7.940,148.642
C08021=1167.718,292.536,-70.600,-176.928,7.943,148.642
C08022=1167.713,292.784,-70.630,-176.926,7.947,148.642
C08023=1167.709,293.032,-70.660,-176.923,7.950,148.642
C08024=1167.705,293.280,-70.690,-176.920,7.953,148.642
C08025=1167.700,293.529,-70.720,-176.918,7.956,148.643
C08026=1167.696,293.777,-70.750,-176.915,7.959,148.642
C08027=1167.692,294.025,-70.779,-176.913,7.962,148.642
C08028=1167.687,294.273,-70.810,-176.910,7.965,148.643
C08029=1167.684,294.522,-70.840,-176.908,7.968,148.643
C08030=1167.680,294.769,-70.870,-176.906,7.970,148.643
C08031=1167.675,295.018,-70.900,-176.903,7.973,148.642
C08032=1167.671,295.266,-70.930,-176.900,7.977,148.643
C08033=1167.667,295.514,-70.960,-176.898,7.980,148.643
C08034=1167.662,295.762,-70.990,-176.895,7.982,148.643
C08035=1167.658,296.010,-71.020,-176.893,7.986,148.643
C08036=1167.653,296.258,-71.051,-176.890,7.989,148.643
C08037=1167.649,296.506,-71.080,-176.887,7.992,148.643
C08038=1167.646,296.755,-71.111,-176.885,7.995,148.643
C08039=1167.641,297.003,-71.141,-176.882,7.998,148.643
C08040=1167.637,297.251,-71.171,-176.879,8.001,148.643
C08041=1167.632,297.499,-71.202,-176.877,8.004,148.643
C08042=1167.628,297.747,-71.231,-176.874,8.007,148.643
C08043=1167.624,297.995,-71.262,-176.872,8.010,148.643
C08044=1167.620,298.243,-71.292,-176.869,8.013,148.643
C08045=1167.615,298.492,-71.322,-176.867,8.016,148.643
C08046=1167.612,298.740,-71.353,-176.864,8.019,148.643
C08047=1167.607,298.988,-71.383,-176.862,8.023,148.643
C08048=1167.603,299.236,-71.413,-176.859,8.026,148.643
C08049=1167.598,299.484,-71.444,-176.856,8.029,148.643
C08050=1167.595,299.732,-71.474,-176.854,8.032,148.643
C08051=1167.590,299.981,-71.504,-176.851,8.035,148.643
C08052=1167.586,300.228,-71.534,-176.848,8.038,148.643
C08053=1167.581,300.476,-71.565,-176.846,8.041,148.644
C08054=1167.578,300.724,-71.595,-176.843,8.044,148.644
C08055=1167.574,300.973,-71.626,-176.841,8.047,148.644
C08056=1167.569,301.221,-71.656,-176.838,8.050,148.644
C08057=1167.565,301.469,-71.687,-176.836,8.053,148.644
C08058=1167.560,301.717,-71.717,-176.833,8.057,148.644
C08059=1167.556,301.965,-71.748,-176.831,8.060,148.644
C08060=1167.552,302.213,-71.779,-176.828,8.063,148.644
C08061=1167.548,302.461,-71.809,-176.825,8.066,148.644
C08062=1167.543,302.709,-71.839,-176.822,8.070,148.644
C08063=1167.539,302.957,-71.870,-176.820,8.073,148.644
C08064=1167.535,303.206,-71.901,-176.817,8.076,148.644
C08065=1167.531,303.454,-71.931,-176.814,8.079,148.644
C08066=1167.526,303.702,-71.962,-176.812,8.082,148.644
C08067=1167.522,303.950,-71.992,-176.809,8.085,148.644
C08068=1167.518,304.198,-72.023,-176.807,8.089,148.644
C08069=1167.514,304.446,-72.054,-176.804,8.092,148.644
C08070=1167.509,304.694,-72.085,-176.802,8.094,148.644
C08071=1167.506,304.942,-72.115,-176.799,8.098,148.645
C08072=1167.501,305.190,-72.146,-176.797,8.101,148.645
C08073=1167.497,305.438,-72.177,-176.794,8.104,148.645
C08074=1167.493,305.687,-72.208,-176.792,8.107,148.645
C08075=1167.489,305.934,-72.238,-176.789,8.110,148.645
C08076=1167.484,306.182,-72.269,-176.786,8.113,148.645
C08077=1167.480,306.431,-72.300,-176.784,8.116,148.645
C08078=1167.476,306.679,-72.331,-176.781,8.120,148.645
C08079=1167.471,306.926,-72.362,-176.779,8.123,148.645
C08080=1167.468,307.175,-72.393,-176.776,8.126,148.645
C08081=1167.463,307.423,-72.423,-176.774,8.129,148.645
C08082=1167.459,307.671,-72.454,-176.771,8.132,148.645
C08083=1167.455,307.919,-72.485,-176.769,8.135,148.645
C08084=1167.450,308.167,-72.516,-176.766,8.138,148.646
C08085=1167.447,308.414,-72.547,-176.764,8.141,148.646
C08086=1167.443,308.663,-72.578,-176.761,8.144,148.646
C08087=1167.438,308.911,-72.609,-176.759,8.148,148.646
C08088=1167.433,309.159,-72.640,-176.755,8.151,148.646
C08089=1167.430,309.407,-72.671,-176.753,8.155,148.646
C08090=1167.425,309.655,-72.702,-176.750,8.158,148.646
C08091=1167.421,309.904,-72.733,-176.748,8.161,148.646
C08092=1167.416,310.151,-72.764,-176.745,8.164,148.646
C08093=1167.413,310.398,-72.795,-176.743,8.167,148.646
C08094=1167.409,310.647,-72.826,-176.740,8.170,148.646
C08095=1167.404,310.895,-72.857,-176.738,8.173,148.646
C08096=1167.401,311.143,-72.889,-176.735,8.176,148.646
C08097=1167.396,311.391,-72.919,-176.733,8.180,148.647
C08098=1167.392,311.640,-72.951,-176.730,8.183,148.647
C08099=1167.388,311.887,-72.982,-176.728,8.186,148.647
C08100=1167.384,312.136,-73.013,-176.725,8.189,148.647
C08101=1167.379,312.383,-73.045,-176.723,8.192,148.647
C08102=1167.375,312.631,-73.075,-176.720,8.195,148.647
C08103=1167.371,312.879,-73.107,-176.718,8.199,148.647
C08104=1167.366,313.127,-73.138,-176.714,8.202,148.647
C08105=1167.362,313.376,-73.169,-176.712,8.206,148.647
C08106=1167.357,313.653,-73.204,-176.709,8.209,148.647
C08107=1167.353,313.929,-73.239,-176.707,8.213,148.648
C08108=1167.349,314.207,-73.275,-176.704,8.216,148.648
C08109=1167.344,314.484,-73.309,-176.701,8.220,148.648
C08110=1167.339,314.731,-73.341,-176.698,8.223,148.648
C08111=1167.336,314.979,-73.373,-176.696,8.226,148.648
C08112=1167.331,315.227,-73.403,-176.693,8.229,148.648
C08113=1167.327,315.475,-73.435,-176.691,8.232,148.648
C08114=1167.323,315.723,-73.466,-176.688,8.235,148.648
C08115=1167.319,315.971,-73.498,-176.686,8.239,148.648
C08116=1167.315,316.219,-73.529,-176.683,8.242,148.648
C08117=1167.310,316.468,-73.561,-176.680,8.246,148.649
C08118=1167.306,316.716,-73.593,-176.678,8.249,148.649
C08119=1167.302,316.963,-73.624,-176.675,8.252,148.649
C08120=1167.298,317.212,-73.655,-176.673,8.255,148.649
C08121=1167.294,317.459,-73.687,-176.670,8.258,148.649
C08122=1167.290,317.707,-73.719,-176.668,8.262,148.649
C08123=1167.285,317.955,-73.749,-176.665,8.265,148.649
C08124=1167.282,318.203,-73.781,-176.663,8.268,148.649
C08125=1167.277,318.451,-73.814,-176.661,8.271,148.649
C08126=1167.273,318.699,-73.845,-176.658,8.274,148.649
C08127=1167.269,318.947,-73.876,-176.655,8.278,148.650
C08128=1167.265,319.195,-73.908,-176.652,8.281,148.650
C08129=1167.261,319.443,-73.940,-176.650,8.285,148.650
C08130=1167.256,319.691,-73.972,-176.647,8.287,148.650
C08131=1167.252,319.939,-74.004,-176.645,8.291,148.650
C08132=1167.248,320.187,-74.035,-176.643,8.294,148.650
C08133=1167.244,320.435,-74.066,-176.640,8.297,148.650
C08134=1167.239,320.683,-74.099,-176.638,8.300,148.650
C08135=1167.236,320.931,-74.131,-176.634,8.304,148.650
C08136=1167.231,321.178,-74.162,-176.632,8.307,148.651
C08137=1167.228,321.426,-74.194,-176.630,8.311,148.651
C08138=1167.223,321.675,-74.226,-176.627,8.314,148.651
C08139=1167.219,321.922,-74.258,-176.625,8.317,148.651
C08140=1167.215,322.170,-74.290,-176.622,8.320,148.651
C08141=1167.211,322.418,-74.322,-176.620,8.323,148.651
C08142=1167.206,322.666,-74.354,-176.617,8.327,148.651
C08143=1167.203,322.914,-74.385,-176.614,8.330,148.651
C08144=1167.198,323.162,-74.418,-176.612,8.334,148.652
C08145=1167.195,323.410,-74.450,-176.610,8.337,148.652
C08146=1167.190,323.657,-74.481,-176.607,8.340,148.652
C08147=1167.186,323.906,-74.514,-176.605,8.343,148.652
C08148=1167.182,324.154,-74.545,-176.602,8.347,148.652
C08149=1167.178,324.401,-74.577,-176.599,8.350,148.652
C08150=1167.173,324.650,-74.609,-176.597,8.353,148.652
C08151=1167.170,324.898,-74.641,-176.594,8.357,148.653
C08152=1167.166,325.146,-74.673,-176.592,8.360,148.653
C08153=1167.161,325.393,-74.706,-176.589,8.363,148.653
C08154=1167.157,325.641,-74.738,-176.587,8.366,148.653
C08155=1167.153,325.889,-74.770,-176.584,8.369,148.653
C08156=1167.149,326.137,-74.802,-176.582,8.373,148.653
C08157=1167.144,326.385,-74.834,-176.580,8.376,148.653
C08158=1167.141,326.633,-74.866,-176.576,8.380,148.654
C08159=1167.136,326.880,-74.899,-176.574,8.383,148.654
C08160=1167.133,327.129,-74.931,-176.572,8.386,148.654
C08161=1167.128,327.376,-74.963,-176.570,8.390,148.654
C08162=1167.124,327.624,-74.995,-176.567,8.393,148.654
C08163=1167.120,327.872,-75.028,-176.565,8.396,148.654
C08164=1167.116,328.120,-75.060,-176.562,8.400,148.655
C08165=1167.111,328.368,-75.092,-176.559,8.403,148.655
C08166=1167.107,328.616,-75.124,-176.557,8.406,148.655
C08167=1167.103,328.863,-75.157,-176.554,8.410,148.655
C08168=1167.100,329.111,-75.189,-176.552,8.413,148.655
C08169=1167.095,329.360,-75.221,-176.549,8.416,148.655
C08170=1167.092,329.607,-75.254,-176.546,8.420,148.655
C08171=1167.087,329.855,-75.286,-176.544,8.423,148.656
C08172=1167.083,330.103,-75.319,-176.542,8.427,148.656
C08173=1167.079,330.351,-75.351,-176.539,8.430,148.656
C08174=1167.074,330.599,-75.383,-176.537,8.433,148.656
C08175=1167.071,330.846,-75.416,-176.535,8.436,148.656
C08176=1167.067,331.095,-75.448,-176.532,8.440,148.656
C08177=1167.062,331.342,-75.481,-176.529,8.443,148.656
C08178=1167.058,331.590,-75.513,-176.527,8.447,148.657
C08179=1167.054,331.838,-75.546,-176.524,8.450,148.657
C08180=1167.050,332.086,-75.578,-176.522,8.453,148.657
C08181=1167.046,332.333,-75.611,-176.519,8.456,148.657
C08182=1167.042,332.582,-75.643,-176.516,8.460,148.657
C08183=1167.038,332.829,-75.677,-176.514,8.464,148.658
C08184=1167.034,333.077,-75.708,-176.512,8.467,148.658
C08185=1167.029,333.324,-75.741,-176.510,8.470,148.658
C08186=1167.025,333.572,-75.774,-176.507,8.473,148.658
C08187=1167.021,333.820,-75.806,-176.504,8.477,148.658
C08188=1167.017,334.068,-75.839,-176.502,8.481,148.658
C08189=1167.013,334.316,-75.872,-176.499,8.484,148.659
C08190=1167.009,334.564,-75.905,-176.497,8.487,148.659
C08191=1167.005,334.811,-75.938,-176.494,8.490,148.659
C08192=1167.001,335.060,-75.970,-176.492,8.494,148.659
C08193=1166.997,335.308,-76.003,-176.489,8.498,148.659
C08194=1166.992,335.555,-76.036,-176.487,8.501,148.659
C08195=1166.989,335.803,-76.068,-176.485,8.504,148.660
C08196=1166.985,336.051,-76.101,-176.482,8.507,148.660
C08197=1166.980,336.299,-76.134,-176.479,8.511,148.660
C08198=1166.976,336.546,-76.168,-176.477,8.515,148.660
C08199=1166.972,336.795,-76.200,-176.474,8.518,148.660
C08200=1166.968,337.042,-76.233,-176.472,8.521,148.661
C08201=1166.964,337.290,-76.266,-176.470,8.524,148.661
C08202=1166.960,337.538,-76.299,-176.467,8.529,148.661
C08203=1166.956,337.785,-76.332,-176.465,8.532,148.661
C08204=1166.952,338.033,-76.365,-176.462,8.535,148.661
C08205=1166.947,338.282,-76.398,-176.460,8.538,148.661
C08206=1166.943,338.529,-76.431,-176.457,8.542,148.662
C08207=1166.940,338.777,-76.463,-176.455,8.546,148.662
C08208=1166.936,339.024,-76.497,-176.452,8.549,148.662
C08209=1166.932,339.272,-76.530,-176.450,8.552,148.662
C08210=1166.926,339.551,-76.567,-176.447,8.556,148.663
C08211=1166.922,339.831,-76.604,-176.444,8.560,148.663
C08212=1166.917,340.110,-76.642,-176.441,8.564,148.663
C08213=1166.912,340.390,-76.679,-176.439,8.568,148.663
C08214=1166.908,340.638,-76.712,-176.436,8.572,148.663
C08215=1166.904,340.886,-76.745,-176.434,8.575,148.664
C08216=1166.900,341.134,-76.778,-176.431,8.578,148.664
C08217=1166.896,341.381,-76.811,-176.429,8.581,148.664
C08218=1166.892,341.629,-76.845,-176.427,8.585,148.664
C08219=1166.888,341.876,-76.878,-176.424,8.589,148.664
C08220=1166.884,342.124,-76.912,-176.421,8.592,148.665
C08221=1166.880,342.372,-76.945,-176.419,8.595,148.665
C08222=1166.876,342.620,-76.978,-176.417,8.599,148.665
C08223=1166.872,342.868,-77.011,-176.414,8.603,148.665
C08224=1166.868,343.115,-77.045,-176.412,8.606,148.665
C08225=1166.864,343.363,-77.078,-176.409,8.609,148.666
C08226=1166.859,343.611,-77.111,-176.407,8.613,148.666
C08227=1166.855,343.859,-77.144,-176.404,8.617,148.666
C08228=1166.851,344.106,-77.178,-176.402,8.620,148.666
C08229=1166.847,344.353,-77.211,-176.400,8.623,148.667
C08230=1166.843,344.601,-77.244,-176.397,8.628,148.667
C08231=1166.840,344.850,-77.278,-176.395,8.631,148.667
C08232=1166.835,345.098,-77.311,-176.392,8.634,148.667
C08233=1166.831,345.345,-77.345,-176.390,8.637,148.667
C08234=1166.827,345.593,-77.379,-176.387,8.642,148.668
C08235=1166.823,345.840,-77.412,-176.385,8.645,148.668
C08236=1166.819,346.088,-77.445,-176.383,8.648,148.668
C08237=1166.815,346.336,-77.479,-176.380,8.651,148.668
C08238=1166.811,346.584,-77.512,-176.377,8.656,148.669
C08239=1166.806,346.832,-77.546,-176.375,8.659,148.669
C08240=1166.802,347.079,-77.580,-176.373,8.662,148.669
C08241=1166.798,347.326,-77.613,-176.370,8.666,148.669
C08242=1166.794,347.574,-77.646,-176.368,8.670,148.670
C08243=1166.791,347.822,-77.680,-176.365,8.673,148.670
C08244=1166.786,348.070,-77.714,-176.363,8.676,148.670
C08245=1166.782,348.317,-77.748,-176.361,8.681,148.670
C08246=1166.778,348.565,-77.781,-176.358,8.684,148.671
C08247=1166.774,348.813,-77.814,-176.356,8.687,148.671
C08248=1166.770,349.061,-77.849,-176.353,8.691,148.671
C08249=1166.766,349.308,-77.882,-176.351,8.695,148.671
C08250=1166.762,349.555,-77.916,-176.349,8.698,148.672
C08251=1166.758,349.803,-77.949,-176.346,8.701,148.672
C08252=1166.754,350.051,-77.984,-176.343,8.705,148.672
C08253=1166.750,350.299,-78.017,-176.341,8.709,148.672
C08254=1166.746,350.546,-78.051,-176.339,8.712,148.673
C08255=1166.741,350.794,-78.085,-176.336,8.716,148.673
C08256=1166.738,351.042,-78.119,-176.334,8.720,148.673
C08257=1166.734,351.289,-78.153,-176.332,8.723,148.673
C08258=1166.730,351.537,-78.186,-176.329,8.727,148.674
C08259=1166.726,351.785,-78.221,-176.327,8.730,148.674
C08260=1166.722,352.033,-78.254,-176.324,8.734,148.674
C08261=1166.717,352.280,-78.289,-176.322,8.738,148.675
C08262=1166.713,352.527,-78.323,-176.320,8.741,148.675
C08263=1166.710,352.776,-78.356,-176.317,8.745,148.675
C08264=1166.705,353.023,-78.391,-176.315,8.749,148.675
C08265=1166.701,353.270,-78.424,-176.312,8.752,148.675
C08266=1166.698,353.519,-78.458,-176.310,8.756,148.676
C08267=1166.693,353.766,-78.492,-176.308,8.760,148.676
C08268=1166.689,354.013,-78.526,-176.305,8.763,148.676
C08269=1166.686,354.261,-78.561,-176.303,8.766,148.677
C08270=1166.681,354.509,-78.594,-176.300,8.770,148.677
C08271=1166.677,354.756,-78.629,-176.298,8.774,148.677
C08272=1166.674,355.004,-78.663,-176.296,8.777,148.677
C08273=1166.669,355.252,-78.697,-176.293,8.781,148.678
C08274=1166.665,355.499,-78.731,-176.291,8.785,148.678
C08275=1166.662,355.747,-78.765,-176.289,8.788,148.678
C08276=1166.657,355.995,-78.799,-176.286,8.793,148.679
C08277=1166.654,356.242,-78.834,-176.284,8.796,148.679
C08278=1166.649,356.490,-78.868,-176.282,8.799,148.679
C08279=1166.645,356.737,-78.902,-176.279,8.804,148.680
C08280=1166.641,356.985,-78.937,-176.277,8.807,148.680
C08281=1166.638,357.232,-78.971,-176.274,8.810,148.680
C08282=1166.634,357.480,-79.005,-176.272,8.815,148.680
C08283=1166.629,357.728,-79.040,-176.270,8.818,148.681
C08284=1166.625,357.975,-79.074,-176.267,8.821,148.681
C08285=1166.621,358.224,-79.108,-176.265,8.826,148.681
C08286=1166.617,358.471,-79.142,-176.263,8.829,148.682
C08287=1166.613,358.719,-79.177,-176.260,8.833,148.682
C08288=1166.609,358.966,-79.210,-176.258,8.837,148.682
C08289=1166.606,359.213,-79.246,-176.256,8.840,148.682
C08290=1166.601,359.461,-79.280,-176.253,8.844,148.683
C08291=1166.598,359.709,-79.315,-176.251,8.848,148.683
C08292=1166.593,359.956,-79.349,-176.249,8.851,148.683
C08293=1166.590,360.204,-79.383,-176.246,8.855,148.684
C08294=1166.586,360.451,-79.418,-176.244,8.859,148.684
C08295=1166.581,360.699,-79.452,-176.241,8.863,148.684
C08296=1166.578,360.947,-79.487,-176.239,8.866,148.685
C08297=1166.573,361.194,-79.521,-176.237,8.870,148.685
C08298=1166.569,361.442,-79.556,-176.235,8.874,148.685
C08299=1166.566,361.689,-79.590,-176.232,8.877,148.686
C08300=1166.562,361.937,-79.625,-176.230,8.882,148.686
C08301=1166.558,362.185,-79.660,-176.228,8.885,148.686
C08302=1166.554,362.432,-79.694,-176.226,8.889,148.687
C08303=1166.550,362.680,-79.729,-176.223,8.893,148.687
C08304=1166.546,362.927,-79.764,-176.221,8.896,148.688
C08305=1166.542,363.175,-79.799,-176.219,8.900,148.688
C08306=1166.538,363.422,-79.833,-176.216,8.904,148.688
C08307=1166.534,363.670,-79.868,-176.214,8.908,148.689
C08308=1166.530,363.917,-79.903,-176.212,8.912,148.689
C08309=1166.526,364.165,-79.938,-176.210,8.915,148.689
C08310=1166.522,364.412,-79.971,-176.207,8.919,148.690
C08311=1166.518,364.660,-80.007,-176.205,8.923,148.690
C08312=1166.514,364.908,-80.042,-176.203,8.927,148.690
C08313=1166.510,365.155,-80.076,-176.201,8.930,148.691
C08314=1166.505,365.438,-80.116,-176.198,8.934,148.691
C08315=1166.501,365.720,-80.156,-176.196,8.939,148.692
C08316=1166.497,366.002,-80.196,-176.193,8.943,148.692
C08317=1166.492,366.284,-80.235,-176.191,8.948,148.693
C08318=1166.488,366.532,-80.270,-176.189,8.951,148.693
C08319=1166.484,366.780,-80.306,-176.187,8.956,148.693
C08320=1166.480,367.027,-80.340,-176.185,8.959,148.694
C08321=1166.476,367.274,-80.376,-176.183,8.963,148.694
C08322=1166.472,367.522,-80.409,-176.180,8.967,148.695
C08323=1166.469,367.769,-80.445,-176.178,8.971,148.695
C08324=1166.465,368.017,-80.480,-176.176,8.974,148.695
C08325=1166.460,368.264,-80.515,-176.175,8.978,148.696
C08326=1166.456,368.512,-80.550,-176.172,8.982,148.696
C08327=1166.453,368.760,-80.585,-176.170,8.986,148.697
C08328=1166.448,369.006,-80.621,-176.168,8.989,148.697
C08329=1166.444,369.255,-80.655,-176.167,8.993,148.698
C08330=1166.441,369.502,-80.691,-176.165,8.998,148.698
C08331=1166.436,369.749,-80.725,-176.163,9.001,148.699
C08332=1166.433,369.997,-80.761,-176.161,9.005,148.699
C08333=1166.429,370.244,-80.796,-176.159,9.009,148.700
C08334=1166.424,370.492,-80.831,-176.157,9.012,148.700
C08335=1166.421,370.739,-80.866,-176.155,9.016,148.700
C08336=1166.417,370.987,-80.902,-176.153,9.021,148.701
C08337=1166.412,371.234,-80.937,-176.151,9.024,148.702
C08338=1166.409,371.482,-80.972,-176.150,9.028,148.702
C08339=1166.405,371.729,-81.008,-176.148,9.032,148.703
C08340=1166.401,371.977,-81.042,-176.146,9.035,148.703
C08341=1166.397,372.224,-81.078,-176.144,9.039,148.703
C08342=1166.393,372.472,-81.113,-176.143,9.043,148.704
C08343=1166.389,372.719,-81.148,-176.141,9.046,148.705
C08344=1166.385,372.967,-81.183,-176.140,9.050,148.705
C08345=1166.381,373.214,-81.219,-176.138,9.054,148.706
C08346=1166.378,373.462,-81.254,-176.136,9.058,148.706
C08347=1166.373,373.708,-81.289,-176.135,9.061,148.707
C08348=1166.370,373.956,-81.325,-176.133,9.065,148.707
C08349=1166.366,374.204,-81.360,-176.132,9.069,148.708
C08350=1166.362,374.452,-81.395,-176.130,9.073,148.708
C08351=1166.358,374.698,-81.431,-176.128,9.077,148.709
C08352=1166.353,374.946,-81.467,-176.127,9.081,148.710
C08353=1166.350,375.194,-81.502,-176.125,9.084,148.710
C08354=1166.346,375.441,-81.538,-176.124,9.088,148.711
C08355=1166.342,375.688,-81.573,-176.122,9.092,148.711
C08356=1166.338,375.935,-81.609,-176.121,9.096,148.712
C08357=1166.334,376.184,-81.643,-176.120,9.099,148.712
C08358=1166.331,376.431,-81.679,-176.118,9.103,148.713
C08359=1166.326,376.679,-81.715,-176.117,9.107,148.713
C08360=1166.322,376.926,-81.750,-176.115,9.110,148.714
C08361=1166.318,377.173,-81.786,-176.114,9.114,148.715
C08362=1166.315,377.421,-81.821,-176.113,9.117,148.715
C08363=1166.311,377.668,-81.857,-176.112,9.121,148.716
C08364=1166.306,377.916,-81.893,-176.110,9.125,148.717
C08365=1166.302,378.163,-81.928,-176.109,9.129,148.717
C08366=1166.299,378.410,-81.964,-176.108,9.133,148.718
C08367=1166.295,378.658,-81.999,-176.107,9.136,148.719
C08368=1166.291,378.905,-82.035,-176.106,9.140,148.719
C08369=1166.287,379.153,-82.071,-176.105,9.143,148.720
C08370=1166.283,379.400,-82.106,-176.103,9.147,148.720
C08371=1166.279,379.647,-82.142,-176.103,9.151,148.721
C08372=1166.276,379.894,-82.178,-176.101,9.155,148.722
C08373=1166.271,380.142,-82.214,-176.101,9.158,148.722
C08374=1166.267,380.390,-82.250,-176.100,9.162,148.723
C08375=1166.264,380.637,-82.285,-176.099,9.165,148.724
C08376=1166.260,380.884,-82.320,-176.097,9.169,148.724
C08377=1166.255,381.132,-82.357,-176.097,9.172,148.725
C08378=1166.251,381.379,-82.392,-176.095,9.176,148.726
C08379=1166.248,381.627,-82.428,-176.095,9.180,148.727
C08380=1166.244,381.874,-82.465,-176.094,9.183,148.727
C08381=1166.240,382.121,-82.500,-176.093,9.187,148.728
C08382=1166.236,382.369,-82.536,-176.092,9.190,148.729
C08383=1166.232,382.616,-82.571,-176.092,9.193,148.729
C08384=1166.228,382.864,-82.607,-176.091,9.196,148.730
C08385=1166.224,383.111,-82.642,-176.090,9.201,148.731
C08386=1166.221,383.358,-82.679,-176.090,9.204,148.732
C08387=1166.216,383.606,-82.715,-176.089,9.207,148.732
C08388=1166.213,383.853,-82.750,-176.088,9.211,148.733
C08389=1166.209,384.101,-82.786,-176.088,9.214,148.734
C08390=1166.205,384.348,-82.823,-176.087,9.217,148.734
C08391=1166.201,384.595,-82.858,-176.086,9.221,148.735
C08392=1166.197,384.842,-82.894,-176.086,9.225,148.736
C08393=1166.193,385.090,-82.930,-176.085,9.228,148.737
C08394=1166.189,385.337,-82.966,-176.085,9.231,148.737
C08395=1166.185,385.585,-83.002,-176.085,9.234,148.738
C08396=1166.181,385.832,-83.038,-176.084,9.237,148.739
C08397=1166.178,386.080,-83.073,-176.084,9.241,148.740
C08398=1166.173,386.327,-83.110,-176.084,9.244,148.740
C08399=1166.170,386.574,-83.146,-176.083,9.248,148.741
C08400=1166.166,386.822,-83.181,-176.082,9.251,148.742
C08401=1166.162,387.069,-83.218,-176.083,9.254,148.743
C08402=1166.158,387.317,-83.254,-176.082,9.257,148.743
C08403=1166.153,387.564,-83.289,-176.082,9.260,148.744
C08404=1166.150,387.811,-83.326,-176.082,9.264,148.745
C08405=1166.146,388.058,-83.361,-176.082,9.266,148.746
C08406=1166.142,388.306,-83.397,-176.081,9.270,148.746
C08407=1166.139,388.553,-83.434,-176.081,9.272,148.747
C08408=1166.134,388.801,-83.470,-176.081,9.276,148.748
C08409=1166.131,389.047,-83.506,-176.081,9.278,148.749
C08410=1166.127,389.295,-83.542,-176.081,9.282,148.749
C08411=1166.123,389.543,-83.578,-176.081,9.284,148.750
C08412=1166.119,389.790,-83.614,-176.081,9.288,148.751
C08413=1166.115,390.037,-83.650,-176.081,9.290,148.752
C08414=1166.112,390.284,-83.686,-176.081,9.293,148.752
C08415=1166.107,390.532,-83.722,-176.081,9.296,148.753
C08416=1166.104,390.780,-83.758,-176.081,9.299,148.754
C08417=1166.099,391.027,-83.795,-176.081,9.302,148.755
C08418=1166.095,391.312,-83.836,-176.081,9.305,148.756
C08419=1166.091,391.597,-83.878,-176.081,9.309,148.757
C08420=1166.086,391.882,-83.919,-176.082,9.312,148.758
C08421=1166.082,392.167,-83.961,-176.081,9.315,148.758
C08422=1166.077,392.415,-83.997,-176.082,9.318,148.759
C08423=1166.074,392.662,-84.033,-176.082,9.321,148.760
C08424=1166.070,392.909,-84.069,-176.082,9.323,148.761
C08425=1166.066,393.157,-84.105,-176.082,9.326,148.761
C08426=1166.063,393.404,-84.142,-176.083,9.329,148.762
C08427=1166.058,393.652,-84.178,-176.083,9.331,148.763
C08428=1166.055,393.899,-84.214,-176.083,9.334,148.764
C08429=1166.050,394.147,-84.250,-176.083,9.336,148.764
C08430=1166.047,394.393,-84.286,-176.084,9.339,148.765
C08431=1166.043,394.641,-84.322,-176.084,9.342,148.766
C08432=1166.039,394.888,-84.359,-176.084,9.344,148.767
C08433=1166.035,395.136,-84.395,-176.084,9.347,148.767
C08434=1166.032,395.383,-84.431,-176.084,9.349,148.768
C08435=1166.027,395.631,-84.467,-176.085,9.352,148.769
C08436=1166.024,395.878,-84.504,-176.085,9.355,148.770
C08437=1166.019,396.125,-84.540,-176.086,9.357,148.770
C08438=1166.016,396.372,-84.576,-176.086,9.359,148.771
C08439=1166.012,396.620,-84.612,-176.086,9.362,148.772
C08440=1166.008,396.867,-84.648,-176.087,9.365,148.773
C08441=1166.004,397.115,-84.685,-176.087,9.366,148.773
C08442=1166.001,397.362,-84.721,-176.087,9.369,148.774
C08443=1165.996,397.609,-84.757,-176.088,9.372,148.775
C08444=1165.993,397.856,-84.793,-176.088,9.374,148.776
C08445=1165.988,398.104,-84.829,-176.089,9.376,148.776
C08446=1165.984,398.351,-84.866,-176.089,9.379,148.777
C08447=1165.981,398.599,-84.902,-176.089,9.381,148.778
C08448=1165.977,398.846,-84.939,-176.090,9.383,148.778
C08449=1165.973,399.093,-84.974,-176.090,9.386,148.779
C08450=1165.969,399.341,-85.011,-176.091,9.388,148.780
C08451=1165.965,399.588,-85.047,-176.091,9.390,148.781
C08452=1165.961,399.835,-85.083,-176.091,9.393,148.781
C08453=1165.958,400.082,-85.120,-176.092,9.395,148.782
C08454=1165.953,400.330,-85.156,-176.092,9.397,148.783
C08455=1165.950,400.577,-85.192,-176.093,9.399,148.783
C08456=1165.946,400.825,-85.228,-176.093,9.401,148.784
C08457=1165.942,401.072,-85.264,-176.094,9.403,148.785
C08458=1165.938,401.319,-85.301,-176.094,9.406,148.786
C08459=1165.934,401.567,-85.337,-176.095,9.408,148.786
C08460=1165.930,401.813,-85.374,-176.095,9.410,148.787
C08461=1165.926,402.061,-85.410,-176.096,9.412,148.788
C08462=1165.923,402.308,-85.446,-176.096,9.415,148.788
C08463=1165.918,402.556,-85.482,-176.097,9.416,148.789
C08464=1165.915,402.803,-85.519,-176.097,9.419,148.790
C08465=1165.910,403.051,-85.555,-176.098,9.421,148.790
C08466=1165.907,403.298,-85.591,-176.098,9.422,148.791
C08467=1165.903,403.545,-85.628,-176.098,9.425,148.792
C08468=1165.899,403.793,-85.664,-176.099,9.427,148.792
C08469=1165.895,404.039,-85.700,-176.099,9.429,148.793
C08470=1165.891,404.287,-85.736,-176.100,9.431,148.794
C08471=1165.887,404.534,-85.773,-176.101,9.433,148.794
C08472=1165.883,404.781,-85.809,-176.101,9.435,148.795
C08473=1165.880,405.029,-85.845,-176.102,9.437,148.796
C08474=1165.876,405.276,-85.882,-176.102,9.439,148.796
C08475=1165.872,405.524,-85.917,-176.102,9.441,148.797
C08476=1165.868,405.771,-85.954,-176.103,9.443,148.798
C08477=1165.864,406.018,-85.991,-176.103,9.445,148.798
C08478=1165.860,406.265,-86.027,-176.103,9.447,148.799
C08479=1165.856,406.513,-86.064,-176.104,9.449,148.800
C08480=1165.853,406.759,-86.100,-176.105,9.451,148.800
C08481=1165.848,407.007,-86.136,-176.105,9.453,148.801
C08482=1165.845,407.254,-86.172,-176.106,9.455,148.802
C08483=1165.840,407.502,-86.208,-176.106,9.456,148.802
C08484=1165.836,407.749,-86.245,-176.107,9.458,148.803
C08485=1165.833,407.996,-86.281,-176.107,9.461,148.803
C08486=1165.829,408.244,-86.318,-176.108,9.463,148.804
C08487=1165.825,408.491,-86.354,-176.108,9.464,148.805
C08488=1165.821,408.738,-86.391,-176.108,9.467,148.805
C08489=1165.817,408.986,-86.427,-176.109,9.468,148.806
C08490=1165.813,409.233,-86.463,-176.109,9.470,148.807
C08491=1165.809,409.480,-86.499,-176.110,9.472,148.807
C08492=1165.806,409.727,-86.536,-176.110,9.474,148.808
C08493=1165.802,409.974,-86.572,-176.111,9.476,148.808
C08494=1165.798,410.222,-86.608,-176.111,9.478,148.809
C08495=1165.794,410.469,-86.645,-176.112,9.479,148.809
C08496=1165.790,410.716,-86.682,-176.112,9.481,148.810
C08497=1165.787,410.965,-86.718,-176.112,9.483,148.811
C08498=1165.783,411.212,-86.754,-176.113,9.485,148.811
C08499=1165.778,411.459,-86.791,-176.113,9.486,148.812
C08500=1165.775,411.706,-86.827,-176.114,9.488,148.813
C08501=1165.771,411.954,-86.864,-176.114,9.490,148.813
C08502=1165.767,412.201,-86.900,-176.114,9.492,148.814
C08503=1165.763,412.448,-86.936,-176.115,9.494,148.814
C08504=1165.759,412.696,-86.973,-176.115,9.495,148.815
C08505=1165.755,412.942,-87.009,-176.116,9.497,148.816
C08506=1165.751,413.190,-87.045,-176.116,9.499,148.816
C08507=1165.748,413.437,-87.082,-176.117,9.501,148.817
C08508=1165.744,413.684,-87.119,-176.117,9.503,148.817
C08509=1165.739,413.932,-87.155,-176.118,9.504,148.818
C08510=1165.736,414.179,-87.191,-176.118,9.507,148.818
C08511=1165.732,414.426,-87.228,-176.118,9.508,148.819
C08512=1165.728,414.674,-87.263,-176.119,9.510,148.820
C08513=1165.724,414.921,-87.300,-176.119,9.512,148.820
C08514=1165.720,415.168,-87.337,-176.120,9.513,148.821
C08515=1165.717,415.416,-87.373,-176.119,9.516,148.821
C08516=1165.714,415.663,-87.409,-176.120,9.517,148.822
C08517=1165.713,415.910,-87.446,-176.120,9.519,148.822
C08518=1165.712,416.230,-87.492,-176.121,9.520,148.823
C08519=1165.713,416.551,-87.539,-176.121,9.523,148.824
C08520=1165.715,416.871,-87.586,-176.122,9.525,148.824
C08521=1165.719,417.189,-87.631,-176.122,9.527,148.825
C08522=1165.298,417.191,-87.677,-176.125,9.538,148.829
C08523=1165.294,416.869,-87.630,-176.125,9.536,148.828
C08524=1165.292,416.545,-87.583,-176.124,9.534,148.827
C08525=1165.291,416.223,-87.537,-176.124,9.531,148.827
C08526=1165.292,415.899,-87.490,-176.123,9.530,148.826
C08527=1165.293,415.652,-87.453,-176.123,9.528,148.825
C08528=1165.295,415.404,-87.417,-176.123,9.527,148.825
C08529=1165.300,415.157,-87.381,-176.122,9.524,148.824
C08530=1165.303,414.910,-87.344,-176.122,9.523,148.824
C08531=1165.307,414.663,-87.307,-176.121,9.521,148.823
C08532=1165.311,414.415,-87.271,-176.121,9.519,148.823
C08533=1165.315,414.168,-87.235,-176.120,9.518,148.822
C08534=1165.319,413.921,-87.198,-176.120,9.515,148.821
C08535=1165.322,413.674,-87.162,-176.120,9.514,148.821
C08536=1165.327,413.426,-87.126,-176.119,9.512,148.820
C08537=1165.331,413.179,-87.089,-176.119,9.510,148.820
C08538=1165.334,412.932,-87.053,-176.118,9.509,148.819
C08539=1165.339,412.684,-87.017,-176.119,9.506,148.819
C08540=1165.342,412.436,-86.979,-176.118,9.505,148.818
C08541=1165.345,412.189,-86.943,-176.117,9.503,148.817
C08542=1165.350,411.942,-86.907,-176.117,9.501,148.817
C08543=1165.353,411.695,-86.871,-176.116,9.500,148.816
C08544=1165.357,411.447,-86.834,-176.116,9.497,148.816
C08545=1165.362,411.200,-86.798,-176.116,9.496,148.815
C08546=1165.365,410.953,-86.761,-176.115,9.494,148.814
C08547=1165.369,410.706,-86.725,-176.114,9.492,148.814
C08548=1165.373,410.458,-86.689,-176.115,9.490,148.813
C08549=1165.377,410.211,-86.652,-176.114,9.488,148.813
C08550=1165.381,409.964,-86.615,-176.113,9.486,148.812
C08551=1165.385,409.716,-86.580,-176.113,9.485,148.811
C08552=1165.389,409.469,-86.543,-176.112,9.483,148.811
C08553=1165.392,409.222,-86.507,-176.112,9.481,148.810
C08554=1165.396,408.974,-86.470,-176.112,9.479,148.809
C08555=1165.401,408.727,-86.434,-176.111,9.477,148.809
C08556=1165.404,408.480,-86.397,-176.111,9.476,148.808
C08557=1165.408,408.232,-86.361,-176.110,9.473,148.808
C08558=1165.412,407.986,-86.325,-176.110,9.471,148.807
C08559=1165.416,407.738,-86.289,-176.109,9.470,148.806
C08560=1165.420,407.491,-86.252,-176.108,9.468,148.806
C08561=1165.423,407.244,-86.216,-176.109,9.466,148.805
C08562=1165.428,406.996,-86.179,-176.108,9.464,148.805
C08563=1165.431,406.749,-86.143,-176.107,9.462,148.804
C08564=1165.435,406.502,-86.106,-176.107,9.460,148.803
C08565=1165.439,406.254,-86.071,-176.106,9.458,148.803
C08566=1165.442,406.006,-86.034,-176.106,9.456,148.802
C08567=1165.447,405.759,-85.997,-176.105,9.454,148.801
C08568=1165.450,405.512,-85.961,-176.105,9.452,148.801
C08569=1165.454,405.265,-85.924,-176.104,9.450,148.800
C08570=1165.458,405.017,-85.889,-176.104,9.449,148.799
C08571=1165.462,404.770,-85.852,-176.104,9.446,148.799
C08572=1165.465,404.523,-85.816,-176.103,9.444,148.798
C08573=1165.470,404.275,-85.780,-176.103,9.442,148.797
C08574=1165.474,404.028,-85.743,-176.102,9.440,148.797
C08575=1165.478,403.780,-85.707,-176.101,9.438,148.796
C08576=1165.482,403.533,-85.670,-176.101,9.436,148.795
C08577=1165.485,403.286,-85.634,-176.101,9.434,148.795
C08578=1165.489,403.039,-85.598,-176.100,9.432,148.794
C08579=1165.493,402.792,-85.562,-176.100,9.430,148.793
C08580=1165.497,402.544,-85.525,-176.099,9.428,148.793
C08581=1165.501,402.297,-85.489,-176.099,9.425,148.792
C08582=1165.505,402.050,-85.452,-176.098,9.423,148.791
C08583=1165.509,401.802,-85.416,-176.098,9.421,148.790
C08584=1165.512,401.555,-85.380,-176.097,9.419,148.790
C08585=1165.517,401.307,-85.344,-176.097,9.416,148.789
C08586=1165.520,401.060,-85.308,-176.096,9.415,148.788
C08587=1165.525,400.813,-85.271,-176.095,9.413,148.788
C08588=1165.528,400.566,-85.235,-176.095,9.410,148.787
C08589=1165.532,400.319,-85.198,-176.095,9.408,148.786
C08590=1165.536,400.071,-85.162,-176.094,9.406,148.786
C08591=1165.540,399.824,-85.126,-176.094,9.403,148.785
C08592=1165.544,399.576,-85.090,-176.093,9.401,148.784
C08593=1165.548,399.329,-85.053,-176.093,9.399,148.783
C08594=1165.552,399.081,-85.017,-176.092,9.397,148.783
C08595=1165.555,398.834,-84.981,-176.092,9.395,148.782
C08596=1165.559,398.587,-84.944,-176.092,9.392,148.781
C08597=1165.563,398.340,-84.909,-176.091,9.390,148.781
C08598=1165.567,398.093,-84.872,-176.091,9.387,148.780
C08599=1165.571,397.845,-84.836,-176.091,9.385,148.779
C08600=1165.575,397.598,-84.799,-176.090,9.383,148.778
C08601=1165.579,397.350,-84.764,-176.090,9.380,148.778
C08602=1165.583,397.103,-84.727,-176.089,9.378,148.777
C08603=1165.587,396.855,-84.691,-176.088,9.376,148.776
C08604=1165.590,396.609,-84.655,-176.088,9.373,148.775
C08605=1165.595,396.361,-84.618,-176.088,9.371,148.775
C08606=1165.598,396.114,-84.582,-176.088,9.368,148.774
C08607=1165.603,395.866,-84.546,-176.087,9.365,148.773
C08608=1165.606,395.619,-84.510,-176.087,9.364,148.772
C08609=1165.610,395.371,-84.474,-176.087,9.361,148.772
C08610=1165.614,395.124,-84.437,-176.086,9.358,148.771
C08611=1165.618,394.877,-84.401,-176.086,9.355,148.770
C08612=1165.621,394.630,-84.365,-176.086,9.353,148.769
C08613=1165.626,394.382,-84.329,-176.086,9.350,148.769
C08614=1165.629,394.135,-84.293,-176.085,9.347,148.768
C08615=1165.634,393.887,-84.256,-176.085,9.345,148.767
C08616=1165.637,393.640,-84.220,-176.085,9.342,148.766
C08617=1165.641,393.393,-84.184,-176.085,9.340,148.766
C08618=1165.645,393.146,-84.148,-176.084,9.337,148.765
C08619=1165.649,392.898,-84.112,-176.084,9.334,148.764
C08620=1165.652,392.651,-84.075,-176.084,9.332,148.763
C08621=1165.657,392.403,-84.039,-176.084,9.329,148.763
C08622=1165.660,392.156,-84.003,-176.083,9.326,148.762
C08623=1165.665,391.871,-83.962,-176.083,9.323,148.761
C08624=1165.669,391.586,-83.920,-176.083,9.320,148.760
C08625=1165.674,391.301,-83.879,-176.083,9.316,148.759
C08626=1165.679,391.016,-83.836,-176.082,9.313,148.758
C08627=1165.682,390.768,-83.800,-176.083,9.310,148.757
C08628=1165.687,390.520,-83.764,-176.083,9.308,148.757
C08629=1165.690,390.273,-83.728,-176.082,9.305,148.756
C08630=1165.694,390.026,-83.693,-176.083,9.302,148.755
C08631=1165.698,389.779,-83.656,-176.082,9.299,148.754
C08632=1165.701,389.531,-83.620,-176.083,9.295,148.754
C08633=1165.706,389.283,-83.584,-176.083,9.293,148.753
C08634=1165.709,389.037,-83.548,-176.082,9.290,148.752
C08635=1165.714,388.789,-83.512,-176.083,9.287,148.751
C08636=1165.717,388.542,-83.475,-176.083,9.284,148.751
C08637=1165.721,388.294,-83.440,-176.083,9.281,148.750
C08638=1165.725,388.047,-83.404,-176.083,9.277,148.749
C08639=1165.729,387.800,-83.368,-176.083,9.275,148.748
C08640=1165.733,387.553,-83.332,-176.083,9.271,148.747
C08641=1165.737,387.305,-83.296,-176.084,9.268,148.747
C08642=1165.740,387.058,-83.260,-176.084,9.265,148.746
C08643=1165.745,386.810,-83.224,-176.084,9.262,148.745
C08644=1165.749,386.563,-83.188,-176.085,9.258,148.744
C08645=1165.753,386.316,-83.151,-176.085,9.255,148.744
C08646=1165.756,386.068,-83.116,-176.085,9.252,148.743
C08647=1165.760,385.821,-83.080,-176.085,9.249,148.742
C08648=1165.764,385.574,-83.043,-176.086,9.246,148.741
C08649=1165.768,385.326,-83.008,-176.086,9.242,148.741
C08650=1165.772,385.078,-82.972,-176.087,9.239,148.740
C08651=1165.775,384.831,-82.935,-176.087,9.236,148.739
C08652=1165.780,384.585,-82.900,-176.088,9.232,148.738
C08653=1165.784,384.337,-82.864,-176.088,9.229,148.738
C08654=1165.788,384.089,-82.828,-176.089,9.226,148.737
C08655=1165.791,383.842,-82.792,-176.090,9.222,148.736
C08656=1165.796,383.595,-82.756,-176.091,9.218,148.736
C08657=1165.799,383.347,-82.720,-176.091,9.215,148.735
C08658=1165.803,383.100,-82.685,-176.091,9.212,148.734
C08659=1165.807,382.852,-82.648,-176.092,9.209,148.733
C08660=1165.811,382.605,-82.613,-176.093,9.204,148.733
C08661=1165.815,382.358,-82.577,-176.094,9.201,148.732
C08662=1165.819,382.110,-82.541,-176.095,9.198,148.731
C08663=1165.823,381.863,-82.506,-176.096,9.194,148.730
C08664=1165.827,381.615,-82.470,-176.096,9.191,148.730
C08665=1165.831,381.368,-82.433,-176.097,9.187,148.729
C08666=1165.834,381.121,-82.398,-176.098,9.183,148.728
C08667=1165.838,380.873,-82.362,-176.099,9.180,148.728
C08668=1165.842,380.626,-82.327,-176.100,9.176,148.727
C08669=1165.847,380.378,-82.291,-176.101,9.173,148.726
C08670=1165.850,380.131,-82.255,-176.102,9.169,148.726
C08671=1165.854,379.883,-82.220,-176.103,9.166,148.725
C08672=1165.857,379.637,-82.183,-176.104,9.162,148.724
C08673=1165.862,379.389,-82.147,-176.105,9.159,148.724
C08674=1165.865,379.141,-82.112,-176.106,9.154,148.723
C08675=1165.870,378.894,-82.077,-176.107,9.151,148.722
C08676=1165.873,378.647,-82.041,-176.108,9.147,148.722
C08677=1165.878,378.399,-82.005,-176.110,9.143,148.721
C08678=1165.881,378.152,-81.969,-176.111,9.140,148.721
C08679=1165.885,377.904,-81.934,-176.112,9.136,148.720
C08680=1165.889,377.657,-81.899,-176.114,9.133,148.719
C08681=1165.894,377.410,-81.862,-176.115,9.128,148.719
C08682=1165.897,377.162,-81.827,-176.115,9.125,148.718
C08683=1165.901,376.915,-81.791,-176.117,9.122,148.718
C08684=1165.905,376.667,-81.756,-176.119,9.118,148.717
C08685=1165.909,376.420,-81.721,-176.120,9.114,148.716
C08686=1165.913,376.173,-81.685,-176.122,9.110,148.716
C08687=1165.917,375.925,-81.649,-176.122,9.107,148.715
C08688=1165.921,375.677,-81.613,-176.124,9.103,148.715
C08689=1165.924,375.430,-81.578,-176.125,9.099,148.714
C08690=1165.929,375.182,-81.543,-176.127,9.095,148.713
C08691=1165.933,374.935,-81.508,-176.129,9.092,148.713
C08692=1165.936,374.687,-81.472,-176.130,9.088,148.712
C08693=1165.940,374.440,-81.437,-176.131,9.084,148.712
C08694=1165.944,374.193,-81.402,-176.133,9.080,148.711
C08695=1165.949,373.945,-81.365,-176.135,9.076,148.711
C08696=1165.952,373.698,-81.330,-176.137,9.073,148.710
C08697=1165.956,373.450,-81.295,-176.138,9.069,148.709
C08698=1165.960,373.203,-81.260,-176.140,9.065,148.709
C08699=1165.964,372.955,-81.224,-176.141,9.061,148.708
C08700=1165.968,372.708,-81.189,-176.143,9.058,148.708
C08701=1165.971,372.460,-81.153,-176.145,9.054,148.707
C08702=1165.976,372.213,-81.119,-176.146,9.050,148.707
C08703=1165.980,371.966,-81.083,-176.148,9.046,148.706
C08704=1165.983,371.718,-81.048,-176.150,9.043,148.706
C08705=1165.988,371.471,-81.012,-176.152,9.038,148.705
C08706=1165.992,371.223,-80.978,-176.154,9.034,148.705
C08707=1165.995,370.976,-80.942,-176.155,9.031,148.704
C08708=1166.000,370.729,-80.907,-176.157,9.027,148.704
C08709=1166.004,370.481,-80.872,-176.159,9.023,148.703
C08710=1166.007,370.233,-80.837,-176.161,9.020,148.703
C08711=1166.011,369.986,-80.801,-176.163,9.015,148.702
C08712=1166.015,369.738,-80.767,-176.165,9.012,148.702
C08713=1166.019,369.491,-80.731,-176.167,9.008,148.702
C08714=1166.024,369.243,-80.697,-176.169,9.004,148.701
C08715=1166.027,368.996,-80.661,-176.170,9.001,148.701
C08716=1166.031,368.748,-80.625,-176.173,8.996,148.700
C08717=1166.036,368.501,-80.591,-176.175,8.993,148.700
C08718=1166.039,368.253,-80.555,-176.177,8.989,148.699
C08719=1166.043,368.005,-80.521,-176.178,8.985,148.699
C08720=1166.047,367.759,-80.485,-176.181,8.981,148.698
C08721=1166.051,367.511,-80.451,-176.183,8.977,148.698
C08722=1166.054,367.263,-80.416,-176.185,8.974,148.698
C08723=1166.059,367.016,-80.381,-176.187,8.969,148.697
C08724=1166.063,366.768,-80.346,-176.189,8.966,148.697
C08725=1166.067,366.521,-80.311,-176.191,8.962,148.696
C08726=1166.071,366.273,-80.276,-176.194,8.958,148.696
C08727=1166.075,365.991,-80.236,-176.196,8.954,148.696
C08728=1166.079,365.709,-80.196,-176.198,8.950,148.695
C08729=1166.084,365.426,-80.157,-176.200,8.946,148.695
C08730=1166.089,365.144,-80.117,-176.203,8.941,148.694
C08731=1166.092,364.897,-80.082,-176.205,8.937,148.694
C08732=1166.096,364.648,-80.047,-176.208,8.934,148.693
C08733=1166.101,364.401,-80.013,-176.209,8.930,148.693
C08734=1166.105,364.154,-79.977,-176.212,8.926,148.693
C08735=1166.109,363.906,-79.943,-176.214,8.922,148.692
C08736=1166.112,363.658,-79.908,-176.217,8.918,148.692
C08737=1166.117,363.411,-79.873,-176.219,8.914,148.692
C08738=1166.121,363.163,-79.838,-176.221,8.911,148.691
C08739=1166.125,362.916,-79.804,-176.223,8.906,148.691
C08740=1166.128,362.669,-79.769,-176.225,8.903,148.691
C08741=1166.132,362.421,-79.734,-176.228,8.899,148.690
C08742=1166.136,362.174,-79.700,-176.230,8.895,148.690
C08743=1166.140,361.925,-79.665,-176.232,8.892,148.689
C08744=1166.145,361.678,-79.631,-176.235,8.888,148.689
C08745=1166.148,361.430,-79.595,-176.237,8.884,148.689
C08746=1166.152,361.183,-79.561,-176.239,8.881,148.688
C08747=1166.156,360.935,-79.527,-176.242,8.877,148.688
C08748=1166.161,360.688,-79.492,-176.244,8.873,148.688
C08749=1166.164,360.440,-79.458,-176.247,8.869,148.688
C08750=1166.168,360.193,-79.423,-176.248,8.865,148.687
C08751=1166.172,359.945,-79.389,-176.251,8.862,148.687
C08752=1166.176,359.697,-79.355,-176.254,8.858,148.687
C08753=1166.181,359.450,-79.320,-176.255,8.854,148.686
C08754=1166.184,359.203,-79.285,-176.258,8.850,148.686
C08755=1166.188,358.955,-79.251,-176.260,8.847,148.685
C08756=1166.191,358.708,-79.217,-176.262,8.843,148.685
C08757=1166.196,358.460,-79.182,-176.265,8.839,148.685
C08758=1166.200,358.212,-79.147,-176.267,8.836,148.685
C08759=1166.204,357.965,-79.113,-176.270,8.832,148.684
C08760=1166.208,357.717,-79.079,-176.272,8.828,148.684
C08761=1166.212,357.470,-79.045,-176.274,8.825,148.684
C08762=1166.217,357.222,-79.011,-176.277,8.821,148.683
C08763=1166.220,356.974,-78.977,-176.279,8.817,148.683
C08764=1166.224,356.726,-78.942,-176.282,8.814,148.683
C08765=1166.228,356.479,-78.908,-176.284,8.810,148.682
C08766=1166.232,356.231,-78.874,-176.286,8.806,148.682
C08767=1166.236,355.984,-78.840,-176.289,8.802,148.682
C08768=1166.240,355.736,-78.805,-176.291,8.799,148.682
C08769=1166.244,355.489,-78.771,-176.293,8.795,148.681
C08770=1166.248,355.240,-78.737,-176.296,8.791,148.681
C08771=1166.252,354.993,-78.703,-176.299,8.788,148.681
C08772=1166.256,354.746,-78.669,-176.300,8.784,148.680
C08773=1166.260,354.498,-78.634,-176.303,8.780,148.680
C08774=1166.264,354.250,-78.600,-176.306,8.777,148.680
C08775=1166.268,354.003,-78.567,-176.308,8.774,148.680
C08776=1166.272,353.754,-78.532,-176.311,8.769,148.679
C08777=1166.276,353.507,-78.498,-176.313,8.766,148.679
C08778=1166.280,353.260,-78.464,-176.315,8.762,148.679
C08779=1166.284,353.012,-78.430,-176.318,8.758,148.679
C08780=1166.288,352.764,-78.396,-176.320,8.755,148.678
C08781=1166.293,352.517,-78.362,-176.322,8.752,148.678
C08782=1166.296,352.269,-78.328,-176.325,8.747,148.678
C08783=1166.300,352.021,-78.294,-176.327,8.744,148.677
C08784=1166.305,351.774,-78.260,-176.329,8.741,148.677
C08785=1166.309,351.526,-78.227,-176.332,8.737,148.677
C08786=1166.312,351.278,-78.192,-176.334,8.733,148.677
C08787=1166.317,351.030,-78.159,-176.337,8.730,148.677
C08788=1166.321,350.783,-78.125,-176.339,8.726,148.676
C08789=1166.324,350.536,-78.091,-176.342,8.722,148.676
C08790=1166.329,350.287,-78.057,-176.344,8.719,148.676
C08791=1166.333,350.040,-78.023,-176.347,8.715,148.675
C08792=1166.337,349.793,-77.990,-176.349,8.712,148.675
C08793=1166.340,349.545,-77.956,-176.351,8.708,148.675
C08794=1166.345,349.297,-77.922,-176.354,8.705,148.675
C08795=1166.349,349.050,-77.888,-176.356,8.701,148.674
C08796=1166.353,348.802,-77.855,-176.358,8.697,148.674
C08797=1166.357,348.553,-77.821,-176.361,8.694,148.674
C08798=1166.361,348.306,-77.787,-176.363,8.690,148.674
C08799=1166.365,348.058,-77.754,-176.366,8.687,148.673
C08800=1166.369,347.811,-77.720,-176.368,8.683,148.673
C08801=1166.373,347.564,-77.687,-176.371,8.679,148.673
C08802=1166.377,347.315,-77.652,-176.373,8.676,148.673
C08803=1166.381,347.068,-77.619,-176.375,8.673,148.672
C08804=1166.385,346.820,-77.585,-176.378,8.669,148.672
C08805=1166.389,346.573,-77.552,-176.381,8.665,148.672
C08806=1166.393,346.325,-77.518,-176.383,8.662,148.672
C08807=1166.398,346.077,-77.485,-176.385,8.659,148.672
C08808=1166.402,345.829,-77.451,-176.388,8.655,148.671
C08809=1166.406,345.582,-77.417,-176.390,8.651,148.671
C08810=1166.410,345.334,-77.384,-176.393,8.648,148.671
C08811=1166.414,345.086,-77.351,-176.395,8.645,148.671
C08812=1166.418,344.839,-77.317,-176.398,8.641,148.670
C08813=1166.422,344.591,-77.284,-176.400,8.637,148.670
C08814=1166.425,344.343,-77.250,-176.402,8.634,148.670
C08815=1166.430,344.095,-77.217,-176.405,8.631,148.670
C08816=1166.434,343.847,-77.183,-176.408,8.627,148.670
C08817=1166.438,343.599,-77.150,-176.410,8.623,148.669
C08818=1166.442,343.352,-77.116,-176.412,8.620,148.669
C08819=1166.446,343.104,-77.083,-176.414,8.617,148.669
C08820=1166.451,342.857,-77.050,-176.417,8.613,148.669
C08821=1166.455,342.609,-77.017,-176.420,8.609,148.668
C08822=1166.459,342.361,-76.984,-176.422,8.606,148.668
C08823=1166.463,342.114,-76.951,-176.424,8.603,148.668
C08824=1166.467,341.865,-76.917,-176.427,8.599,148.668
C08825=1166.471,341.617,-76.884,-176.429,8.595,148.668
C08826=1166.475,341.370,-76.851,-176.432,8.592,148.667
C08827=1166.479,341.122,-76.818,-176.434,8.589,148.667
C08828=1166.483,340.874,-76.785,-176.437,8.585,148.667
C08829=1166.487,340.626,-76.751,-176.439,8.581,148.667
C08830=1166.491,340.379,-76.718,-176.441,8.578,148.666
C08831=1166.496,340.099,-76.681,-176.444,8.574,148.666
C08832=1166.501,339.820,-76.643,-176.447,8.570,148.666
C08833=1166.505,339.540,-76.606,-176.450,8.566,148.666
C08834=1166.510,339.261,-76.568,-176.453,8.563,148.666
C08835=1166.514,339.014,-76.536,-176.456,8.558,148.665
C08836=1166.518,338.766,-76.503,-176.458,8.555,148.665
C08837=1166.522,338.518,-76.470,-176.460,8.552,148.665
C08838=1166.526,338.271,-76.436,-176.462,8.549,148.665
C08839=1166.531,338.022,-76.404,-176.465,8.545,148.665
C08840=1166.535,337.774,-76.371,-176.468,8.541,148.664
C08841=1166.539,337.527,-76.338,-176.470,8.538,148.664
C08842=1166.543,337.279,-76.305,-176.472,8.535,148.664
C08843=1166.546,337.032,-76.272,-176.475,8.532,148.664
C08844=1166.551,336.784,-76.239,-176.478,8.528,148.664
C08845=1166.555,336.535,-76.206,-176.480,8.524,148.663
C08846=1166.559,336.288,-76.173,-176.482,8.521,148.663
C08847=1166.563,336.040,-76.140,-176.485,8.518,148.663
C08848=1166.567,335.793,-76.108,-176.487,8.514,148.663
C08849=1166.571,335.544,-76.075,-176.490,8.510,148.663
C08850=1166.575,335.297,-76.042,-176.493,8.507,148.663
C08851=1166.579,335.049,-76.009,-176.495,8.504,148.662
C08852=1166.584,334.800,-75.976,-176.497,8.501,148.662
C08853=1166.587,334.553,-75.944,-176.500,8.497,148.662
C08854=1166.591,334.305,-75.911,-176.502,8.493,148.662
C08855=1166.596,334.057,-75.878,-176.505,8.490,148.662
C08856=1166.600,333.809,-75.845,-176.507,8.487,148.662
C08857=1166.603,333.562,-75.812,-176.510,8.484,148.661
C08858=1166.608,333.313,-75.780,-176.512,8.480,148.661
C08859=1166.612,333.066,-75.747,-176.515,8.476,148.661
C08860=1166.616,332.818,-75.715,-176.517,8.473,148.661
C08861=1166.620,332.571,-75.682,-176.520,8.470,148.661
C08862=1166.625,332.322,-75.650,-176.522,8.467,148.660
C08863=1166.628,332.075,-75.617,-176.524,8.463,148.660
C08864=1166.633,331.827,-75.585,-176.527,8.459,148.660
C08865=1166.637,331.579,-75.552,-176.530,8.456,148.660
C08866=1166.641,331.331,-75.520,-176.532,8.453,148.660
C08867=1166.645,331.083,-75.487,-176.535,8.450,148.660
C08868=1166.650,330.835,-75.455,-176.537,8.446,148.659
C08869=1166.653,330.588,-75.422,-176.540,8.442,148.659
C08870=1166.658,330.340,-75.390,-176.542,8.439,148.659
C08871=1166.661,330.092,-75.357,-176.545,8.436,148.659
C08872=1166.665,329.844,-75.325,-176.547,8.433,148.659
C08873=1166.670,329.596,-75.292,-176.549,8.429,148.659
C08874=1166.674,329.349,-75.260,-176.552,8.426,148.659
C08875=1166.678,329.100,-75.227,-176.555,8.422,148.658
C08876=1166.682,328.852,-75.196,-176.557,8.419,148.658
C08877=1166.686,328.605,-75.162,-176.560,8.416,148.658
C08878=1166.690,328.357,-75.131,-176.562,8.413,148.658
C08879=1166.695,328.109,-75.099,-176.564,8.410,148.658
C08880=1166.698,327.862,-75.066,-176.567,8.406,148.658
C08881=1166.703,327.613,-75.034,-176.570,8.402,148.658
C08882=1166.706,327.365,-75.002,-176.572,8.399,148.657
C08883=1166.711,327.117,-74.969,-176.575,8.396,148.657
C08884=1166.715,326.870,-74.937,-176.577,8.393,148.657
C08885=1166.719,326.622,-74.905,-176.580,8.390,148.657
C08886=1166.723,326.374,-74.873,-176.582,8.386,148.657
C08887=1166.727,326.125,-74.840,-176.585,8.382,148.656
C08888=1166.731,325.879,-74.808,-176.588,8.379,148.656
C08889=1166.736,325.630,-74.776,-176.590,8.376,148.656
C08890=1166.740,325.382,-74.744,-176.592,8.373,148.656
C08891=1166.744,325.134,-74.711,-176.595,8.370,148.656
C08892=1166.748,324.887,-74.680,-176.597,8.366,148.656
C08893=1166.752,324.639,-74.648,-176.599,8.363,148.656
C08894=1166.757,324.390,-74.616,-176.603,8.359,148.656
C08895=1166.760,324.142,-74.584,-176.605,8.356,148.655
C08896=1166.765,323.895,-74.551,-176.607,8.353,148.655
C08897=1166.769,323.647,-74.519,-176.610,8.350,148.655
C08898=1166.772,323.399,-74.487,-176.612,8.346,148.655
C08899=1166.777,323.151,-74.455,-176.615,8.343,148.655
C08900=1166.781,322.903,-74.423,-176.617,8.340,148.655
C08901=1166.785,322.655,-74.392,-176.620,8.336,148.655
C08902=1166.789,322.407,-74.359,-176.623,8.333,148.654
C08903=1166.794,322.160,-74.328,-176.625,8.330,148.654
C08904=1166.797,321.912,-74.296,-176.628,8.326,148.654
C08905=1166.801,321.664,-74.264,-176.630,8.323,148.654
C08906=1166.806,321.416,-74.232,-176.633,8.320,148.654
C08907=1166.810,321.167,-74.201,-176.635,8.317,148.654
C08908=1166.814,320.919,-74.169,-176.638,8.314,148.654
C08909=1166.819,320.672,-74.137,-176.641,8.310,148.654
C08910=1166.823,320.424,-74.105,-176.643,8.306,148.653
C08911=1166.827,320.176,-74.073,-176.646,8.303,148.653
C08912=1166.831,319.928,-74.042,-176.648,8.300,148.653
C08913=1166.835,319.680,-74.009,-176.651,8.297,148.653
C08914=1166.839,319.432,-73.978,-176.653,8.294,148.653
C08915=1166.843,319.184,-73.947,-176.655,8.291,148.653
C08916=1166.847,318.936,-73.915,-176.658,8.288,148.653
C08917=1166.851,318.688,-73.883,-176.661,8.284,148.653
C08918=1166.856,318.440,-73.851,-176.664,8.281,148.653
C08919=1166.860,318.193,-73.819,-176.666,8.277,148.652
C08920=1166.864,317.944,-73.788,-176.669,8.274,148.652
C08921=1166.868,317.696,-73.756,-176.671,8.271,148.652
C08922=1166.872,317.449,-73.725,-176.673,8.268,148.652
C08923=1166.876,317.200,-73.694,-176.676,8.265,148.652
C08924=1166.881,316.952,-73.662,-176.678,8.261,148.652
C08925=1166.885,316.704,-73.630,-176.681,8.258,148.652
C08926=1166.889,316.456,-73.599,-176.683,8.255,148.652
C08927=1166.893,316.208,-73.567,-176.686,8.251,148.652
C08928=1166.897,315.961,-73.536,-176.689,8.248,148.652
C08929=1166.901,315.712,-73.505,-176.691,8.245,148.651
C08930=1166.905,315.464,-73.473,-176.694,8.242,148.651
C08931=1166.909,315.217,-73.441,-176.696,8.238,148.651
C08932=1166.914,314.968,-73.410,-176.699,8.236,148.651
C08933=1166.918,314.721,-73.379,-176.701,8.232,148.651
C08934=1166.922,314.472,-73.348,-176.704,8.229,148.651
C08935=1166.927,314.196,-73.312,-176.707,8.225,148.651
C08936=1166.932,313.919,-73.277,-176.709,8.222,148.651
C08937=1166.937,313.642,-73.242,-176.712,8.218,148.651
C08938=1166.940,313.364,-73.208,-176.715,8.215,148.651
C08939=1166.945,313.117,-73.176,-176.718,8.211,148.650
C08940=1166.949,312.869,-73.145,-176.721,8.208,148.650
C08941=1166.953,312.621,-73.113,-176.723,8.205,148.650
C08942=1166.958,312.373,-73.083,-176.726,8.202,148.650
C08943=1166.961,312.125,-73.051,-176.728,8.198,148.650
C08944=1166.966,311.877,-73.020,-176.731,8.195,148.650
C08945=1166.970,311.628,-72.989,-176.733,8.192,148.650
C08946=1166.974,311.381,-72.957,-176.736,8.189,148.650
C08947=1166.978,311.132,-72.926,-176.738,8.186,148.650
C08948=1166.983,310.885,-72.895,-176.741,8.183,148.650
C08949=1166.987,310.636,-72.864,-176.743,8.180,148.649
C08950=1166.991,310.388,-72.833,-176.746,8.177,148.649
C08951=1166.996,310.140,-72.802,-176.748,8.173,148.649
C08952=1167.000,309.892,-72.770,-176.751,8.170,148.649
C08953=1167.004,309.644,-72.740,-176.754,8.166,148.649
C08954=1167.008,309.396,-72.708,-176.756,8.163,148.649
C08955=1167.012,309.149,-72.678,-176.759,8.160,148.649
C08956=1167.016,308.901,-72.647,-176.761,8.157,148.649
C08957=1167.020,308.652,-72.616,-176.764,8.154,148.649
C08958=1167.025,308.404,-72.585,-176.767,8.151,148.649
C08959=1167.029,308.156,-72.553,-176.769,8.148,148.649
C08960=1167.033,307.908,-72.522,-176.772,8.144,148.649
C08961=1167.038,307.660,-72.492,-176.774,8.142,148.649
C08962=1167.041,307.412,-72.461,-176.777,8.138,148.648
C08963=1167.046,307.164,-72.430,-176.779,8.135,148.648
C08964=1167.050,306.916,-72.399,-176.782,8.132,148.648
C08965=1167.054,306.667,-72.368,-176.784,8.129,148.648
C08966=1167.059,306.420,-72.337,-176.787,8.126,148.648
C08967=1167.063,306.172,-72.307,-176.789,8.123,148.648
C08968=1167.067,305.923,-72.276,-176.792,8.119,148.648
C08969=1167.071,305.675,-72.245,-176.794,8.116,148.648
C08970=1167.076,305.428,-72.214,-176.797,8.113,148.648
C08971=1167.079,305.179,-72.184,-176.800,8.109,148.648
C08972=1167.084,304.931,-72.153,-176.803,8.106,148.648
C08973=1167.088,304.683,-72.122,-176.805,8.103,148.648
C08974=1167.092,304.436,-72.092,-176.808,8.100,148.648
C08975=1167.096,304.187,-72.061,-176.811,8.097,148.648
C08976=1167.101,303.939,-72.030,-176.813,8.094,148.647
C08977=1167.106,303.691,-71.999,-176.816,8.091,148.647
C08978=1167.109,303.443,-71.969,-176.818,8.088,148.647
C08979=1167.113,303.195,-71.938,-176.821,8.085,148.647
C08980=1167.118,302.947,-71.907,-176.823,8.081,148.647
C08981=1167.122,302.699,-71.877,-176.826,8.078,148.647
C08982=1167.126,302.450,-71.846,-176.828,8.075,148.647
C08983=1167.131,302.202,-71.816,-176.831,8.072,148.647
C08984=1167.135,301.954,-71.786,-176.833,8.069,148.647
C08985=1167.139,301.706,-71.755,-176.836,8.066,148.647
C08986=1167.143,301.458,-71.724,-176.838,8.063,148.647
C08987=1167.147,301.210,-71.694,-176.841,8.060,148.647
C08988=1167.152,300.962,-71.663,-176.843,8.057,148.647
C08989=1167.156,300.714,-71.633,-176.846,8.054,148.647
C08990=1167.161,300.466,-71.603,-176.849,8.051,148.647
C08991=1167.164,300.217,-71.572,-176.851,8.047,148.647
C08992=1167.169,299.969,-71.541,-176.854,8.044,148.647
C08993=1167.172,299.722,-71.511,-176.856,8.041,148.646
C08994=1167.177,299.473,-71.481,-176.859,8.038,148.646
C08995=1167.181,299.226,-71.451,-176.862,8.035,148.646
C08996=1167.185,298.977,-71.420,-176.864,8.032,148.646
C08997=1167.190,298.728,-71.390,-176.867,8.029,148.646
C08998=1167.194,298.481,-71.360,-176.870,8.026,148.646
C08999=1167.199,298.233,-71.329,-176.872,8.023,148.646
C09000=1167.203,297.984,-71.299,-176.875,8.020,148.646
C09001=1167.207,297.737,-71.269,-176.877,8.017,148.646
C09002=1167.211,297.488,-71.238,-176.880,8.013,148.646
C09003=1167.215,297.240,-71.209,-176.882,8.010,148.646
C09004=1167.219,296.992,-71.178,-176.885,8.007,148.646
C09005=1167.224,296.744,-71.148,-176.887,8.004,148.646
C09006=1167.228,296.496,-71.118,-176.890,8.001,148.646
C09007=1167.232,296.248,-71.087,-176.893,7.998,148.646
C09008=1167.237,295.999,-71.057,-176.895,7.995,148.646
C09009=1167.240,295.751,-71.027,-176.898,7.992,148.646
C09010=1167.245,295.503,-70.997,-176.901,7.989,148.646
C09011=1167.249,295.255,-70.967,-176.903,7.986,148.646
C09012=1167.253,295.007,-70.937,-176.906,7.983,148.646
C09013=1167.257,294.759,-70.907,-176.908,7.980,148.646
C09014=1167.262,294.510,-70.877,-176.911,7.976,148.646
C09015=1167.266,294.263,-70.847,-176.913,7.973,148.646
C09016=1167.270,294.015,-70.817,-176.916,7.970,148.646
C09017=1167.275,293.766,-70.787,-176.919,7.968,148.646
C09018=1167.279,293.518,-70.757,-176.921,7.964,148.645
C09019=1167.283,293.269,-70.727,-176.924,7.961,148.646
C09020=1167.287,293.021,-70.697,-176.927,7.958,148.646
C09021=1167.291,292.773,-70.667,-176.929,7.955,148.645
C09022=1167.296,292.525,-70.638,-176.932,7.952,148.645
C09023=1167.300,292.277,-70.607,-176.935,7.949,148.645
C09024=1167.304,292.029,-70.577,-176.937,7.946,148.645
C09025=1167.308,291.780,-70.548,-176.940,7.943,148.645
C09026=1167.312,291.533,-70.518,-176.942,7.940,148.645
C09027=1167.317,291.284,-70.488,-176.945,7.937,148.645
C09028=1167.321,291.036,-70.458,-176.947,7.934,148.645
C09029=1167.325,290.788,-70.428,-176.950,7.931,148.645
C09030=1167.330,290.540,-70.399,-176.953,7.928,148.645
C09031=1167.334,290.291,-70.369,-176.956,7.925,148.645
C09032=1167.339,290.043,-70.339,-176.957,7.922,148.645
C09033=1167.342,289.795,-70.309,-176.960,7.919,148.645
C09034=1167.347,289.547,-70.280,-176.963,7.916,148.645
C09035=1167.351,289.299,-70.250,-176.966,7.913,148.645
C09036=1167.356,289.050,-70.220,-176.968,7.910,148.645
C09037=1167.360,288.802,-70.191,-176.971,7.907,148.645
C09038=1167.364,288.554,-70.161,-176.973,7.904,148.645
C09039=1167.369,288.279,-70.128,-176.977,7.900,148.645
C09040=1167.373,288.004,-70.096,-176.979,7.897,148.645
C09041=1167.378,287.730,-70.063,-176.982,7.894,148.645
C09042=1167.383,287.455,-70.030,-176.985,7.890,148.645
C09043=1167.387,287.206,-70.001,-176.988,7.887,148.645
C09044=1167.392,286.958,-69.971,-176.990,7.884,148.645
C09045=1167.395,286.710,-69.941,-176.993,7.881,148.645
C09046=1167.400,286.462,-69.912,-176.995,7.879,148.645
C09047=1167.404,286.213,-69.882,-176.998,7.876,148.645
C09048=1167.409,285.965,-69.852,-177.000,7.873,148.645
C09049=1167.413,285.717,-69.823,-177.003,7.870,148.645
C09050=1167.417,285.469,-69.793,-177.005,7.867,148.645
C09051=1167.421,285.220,-69.764,-177.008,7.864,148.645
C09052=1167.426,284.972,-69.735,-177.011,7.861,148.645
C09053=1167.430,284.724,-69.706,-177.014,7.858,148.645
C09054=1167.435,284.476,-69.677,-177.016,7.855,148.645
C09055=1167.439,284.227,-69.647,-177.019,7.851,148.645
C09056=1167.443,283.979,-69.618,-177.022,7.849,148.645
C09057=1167.447,283.731,-69.588,-177.024,7.846,148.645
C09058=1167.451,283.483,-69.559,-177.027,7.843,148.645
C09059=1167.456,283.235,-69.530,-177.030,7.840,148.645
C09060=1167.460,282.987,-69.500,-177.031,7.837,148.645
C09061=1167.465,282.738,-69.471,-177.034,7.834,148.645
C09062=1167.469,282.490,-69.442,-177.037,7.831,148.645
C09063=1167.473,282.241,-69.413,-177.040,7.828,148.645
C09064=1167.477,281.993,-69.383,-177.042,7.825,148.645
C09065=1167.482,281.746,-69.354,-177.045,7.822,148.645
C09066=1167.486,281.497,-69.326,-177.048,7.819,148.645
C09067=1167.490,281.249,-69.296,-177.050,7.816,148.645
C09068=1167.494,281.000,-69.267,-177.053,7.813,148.645
C09069=1167.498,280.752,-69.238,-177.056,7.810,148.645
C09070=1167.504,280.504,-69.209,-177.058,7.807,148.645
C09071=1167.508,280.256,-69.180,-177.061,7.804,148.645
C09072=1167.512,280.007,-69.150,-177.063,7.802,148.645
C09073=1167.516,279.759,-69.121,-177.066,7.799,148.645
C09074=1167.520,279.511,-69.093,-177.068,7.796,148.645
C09075=1167.525,279.263,-69.064,-177.071,7.793,148.645
C09076=1167.529,279.014,-69.035,-177.074,7.790,148.645
C09077=1167.533,278.766,-69.005,-177.077,7.787,148.645
C09078=1167.537,278.518,-68.976,-177.079,7.784,148.645
C09079=1167.543,278.269,-68.948,-177.082,7.781,148.645
C09080=1167.546,278.021,-68.919,-177.084,7.778,148.645
C09081=1167.551,277.773,-68.890,-177.087,7.776,148.645
C09082=1167.555,277.524,-68.860,-177.089,7.773,148.645
C09083=1167.559,277.277,-68.831,-177.092,7.770,148.645
C09084=1167.563,277.028,-68.803,-177.095,7.767,148.645
C09085=1167.567,276.780,-68.774,-177.098,7.764,148.645
C09086=1167.572,276.531,-68.745,-177.100,7.761,148.645
C09087=1167.577,276.283,-68.716,-177.103,7.757,148.645
C09088=1167.580,276.035,-68.688,-177.105,7.754,148.645
C09089=1167.585,275.787,-68.658,-177.108,7.751,148.645
C09090=1167.590,275.538,-68.630,-177.110,7.749,148.645
C09091=1167.593,275.290,-68.602,-177.113,7.746,148.645
C09092=1167.598,275.042,-68.572,-177.116,7.743,148.646
C09093=1167.602,274.793,-68.544,-177.119,7.740,148.646
C09094=1167.606,274.545,-68.515,-177.121,7.737,148.646
C09095=1167.611,274.297,-68.486,-177.124,7.734,148.646
C09096=1167.615,274.048,-68.458,-177.127,7.732,148.646
C09097=1167.619,273.800,-68.429,-177.129,7.728,148.646
C09098=1167.624,273.552,-68.400,-177.131,7.726,148.646
C09099=1167.629,273.303,-68.372,-177.134,7.723,148.646
C09100=1167.632,273.055,-68.343,-177.137,7.720,148.646
C09101=1167.637,272.806,-68.315,-177.140,7.717,148.646
C09102=1167.642,272.558,-68.286,-177.142,7.714,148.646
C09103=1167.645,272.310,-68.257,-177.145,7.711,148.646
C09104=1167.650,272.061,-68.229,-177.148,7.708,148.646
C09105=1167.654,271.814,-68.201,-177.150,7.706,148.646
C09106=1167.659,271.565,-68.172,-177.153,7.703,148.646
C09107=1167.663,271.317,-68.144,-177.156,7.700,148.646
C09108=1167.667,271.069,-68.115,-177.158,7.697,148.646
C09109=1167.672,270.820,-68.086,-177.161,7.694,148.646
C09110=1167.676,270.572,-68.058,-177.164,7.691,148.646
C09111=1167.680,270.323,-68.030,-177.167,7.688,148.646
C09112=1167.684,270.076,-68.001,-177.168,7.686,148.646
C09113=1167.689,269.827,-67.972,-177.171,7.683,148.646
C09114=1167.693,269.578,-67.944,-177.174,7.680,148.646
C09115=1167.698,269.330,-67.916,-177.177,7.677,148.646
C09116=1167.702,269.081,-67.888,-177.179,7.674,148.646
C09117=1167.707,268.833,-67.859,-177.182,7.671,148.646
C09118=1167.710,268.585,-67.831,-177.184,7.669,148.647
C09119=1167.715,268.336,-67.803,-177.187,7.666,148.647
C09120=1167.719,268.088,-67.775,-177.190,7.663,148.647
C09121=1167.724,267.840,-67.746,-177.192,7.660,148.647
C09122=1167.728,267.592,-67.717,-177.195,7.657,148.647
C09123=1167.732,267.344,-67.690,-177.198,7.654,148.647
C09124=1167.737,267.095,-67.661,-177.200,7.652,148.647
C09125=1167.741,266.847,-67.633,-177.203,7.649,148.647
C09126=1167.745,266.598,-67.604,-177.206,7.646,148.647
C09127=1167.750,266.350,-67.577,-177.208,7.643,148.647
C09128=1167.754,266.101,-67.549,-177.211,7.640,148.647
C09129=1167.759,265.853,-67.521,-177.213,7.638,148.647
C09130=1167.763,265.604,-67.493,-177.216,7.635,148.647
C09131=1167.768,265.356,-67.464,-177.219,7.632,148.647
C09132=1167.771,265.108,-67.436,-177.222,7.629,148.647
C09133=1167.776,264.860,-67.408,-177.224,7.626,148.647
C09134=1167.780,264.611,-67.380,-177.227,7.623,148.647
C09135=1167.785,264.363,-67.352,-177.229,7.621,148.648
C09136=1167.788,264.114,-67.324,-177.232,7.618,148.648
C09137=1167.794,263.866,-67.296,-177.235,7.615,148.648
C09138=1167.798,263.617,-67.268,-177.238,7.612,148.648
C09139=1167.802,263.369,-67.240,-177.240,7.609,148.648
C09140=1167.807,263.121,-67.212,-177.242,7.607,148.648
C09141=1167.811,262.872,-67.184,-177.245,7.604,148.648
C09142=1167.815,262.624,-67.157,-177.248,7.601,148.648
C09143=1167.820,262.351,-67.125,-177.251,7.599,148.648
C09144=1167.824,262.078,-67.094,-177.254,7.596,148.648
C09145=1167.829,261.805,-67.064,-177.257,7.592,148.648
